KUKA KRL program: EPS_2_251825_SA15_A_20260116064058.src

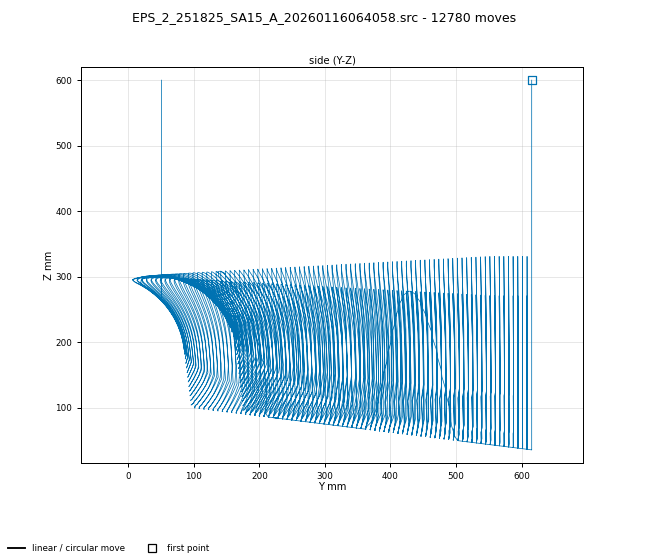
[picture p0: tool path of EPS_2_251825_SA15_A_20260116064058.src, 12780 of 12782 moves have a stored position in this frame; points joined in program order, loops and branches not executed]
&ACCESS RVP
&REL 4
&COMMENT QRS 19112012
&PARAM EDITMASK = *
DEF PART()
EXT BAS (BAS_COMMAND :IN,REAL :IN )
INT I
BAS (#INITMOV,0 )

;KUKA QRS Post kuka4.cps  Date:22-06-2017 !

File_ID=2977

QRS_PRE_INIT()

;Init var - Until changes are made in qrs_pre_init
Outlet_Square_prg=0
Inlet_1_Square_prg=0
Inlet_2_Square_prg=0
Inlet_3_Square_prg=0
Inlet_4_Square_prg=0
Inlet_5_Square_prg=0

Outlet_1={X 0.000, Y 551.740, Z 230.500, B 0.000, E1 0.000 }
Inlet_1={X 0.000, Y 556.010, Z 170.500, B 0.000, E1 166.000 }
Outlet_1_type=201
Inlet_1_type=201
;QRS#1=Sidecore dimensions
;QRS#2=200-8" PVC SDR 35
;QRS#3=200-8" PVC SDR 35
;QRS#4=
;QRS#5=
;QRS#6=
;QRS#7=
;QRS#8=
;QRS#9=12-08 PSX
;QRS#10=12-08 PSX
;QRS#11=
;QRS#12=
;QRS#13=
;QRS#14=
;QRS#15=
;QRS#16=1220x127x610 2'
;QRS#17=EPS Height
;QRS#18=331
;QRS#19=*
;QRS#20= UPDATED VERSION 22-06-2017
;QRS#21=*
Outlet_Square=0100
Inlet_1_Square=0100
Inlet_2_Square=0
Inlet_3_Square=0
Inlet_4_Square=0
Inlet_5_Square=0
Mill_Square=1
Outlet_Square_Prg=204
Inlet_1_Square_prg=204

QRS_INIT()

$ADVANCE=5

; T1
PTP {E1 173.614,E2 173.614}
PTP {X 0,Y 615.487,A -85,B 0,C 180,E1 173.614,E2 173.614,E3 0,E4 0,E5 0,E6 0}
QRS_SPEED_INIT()
LIN {X 0,Y 615.487,Z 600,A -85,B 0,C 180,E1 173.614,E2 173.614,E3 0,E4 0,E5 0,E6 0} C_VEL
LIN {X 0,Y 615.487,Z 45.866,A -85,B 0,C 180,E1 173.614,E2 173.614} C_VEL
LIN {X 0,Y 615.487,Z 37.686,A -85,B 0,C 180,E1 173.614,E2 173.614} C_VEL
LIN {X 0,Y 615.477,Z 35.686,A -85,B 0,C 180,E1 173.428,E2 173.428} C_VEL
LIN {X 0,Y 615.493,Z 35.696,A -85,B 0,C 180,E1 170.801,E2 170.801} C_VEL
LIN {X 0,Y 615.458,Z 35.693,A -85,B 0,C 180,E1 168.138,E2 168.138} C_VEL
LIN {X 0,Y 615.491,Z 35.686,A -85,B 0,C 180,E1 165.451,E2 165.451} C_VEL
LIN {X 0,Y 615.474,Z 35.697,A -85,B 0,C 180,E1 162.729,E2 162.729} C_VEL
LIN {X 0,Y 615.471,Z 35.688,A -85,B 0,C 180,E1 159.966,E2 159.966} C_VEL
LIN {X 0,Y 615.486,Z 35.701,A -85,B 0,C 180,E1 157.155,E2 157.155} C_VEL
LIN {X 0,Y 615.454,Z 35.691,A -85,B 0,C 180,E1 154.437,E2 154.437} C_VEL
LIN {X 0,Y 615.494,Z 35.698,A -85,B 0,C 180,E1 151.548,E2 151.548} C_VEL
LIN {X 0,Y 615.45,Z 35.694,A -85,B 0,C 180,E1 148.919,E2 148.919} C_VEL
LIN {X 0,Y 615.464,Z 35.69,A -85,B 0,C 180,E1 146.469,E2 146.469} C_VEL
LIN {X 0,Y 615.474,Z 35.698,A -85,B 0,C 180,E1 143.574,E2 143.574} C_VEL
LIN {X 0,Y 615.447,Z 35.693,A -85,B 0,C 180,E1 140.942,E2 140.942} C_VEL
LIN {X 0,Y 615.48,Z 35.69,A -85,B 0,C 180,E1 138.525,E2 138.525} C_VEL
LIN {X 0,Y 615.468,Z 35.698,A -85,B 0,C 180,E1 135.848,E2 135.848} C_VEL
LIN {X 0,Y 615.441,Z 35.694,A -85,B 0,C 180,E1 133.248,E2 133.248} C_VEL
LIN {X 0,Y 615.488,Z 35.694,A -85,B 0,C 180,E1 130.606,E2 130.606} C_VEL
LIN {X 0,Y 615.451,Z 35.698,A -85,B 0,C 180,E1 128.007,E2 128.007} C_VEL
LIN {X 0,Y 615.435,Z 35.695,A -85,B 0,C 180,E1 125.619,E2 125.619} C_VEL
LIN {X 0,Y 615.458,Z 35.694,A -85,B 0,C 180,E1 123.238,E2 123.238} C_VEL
LIN {X 0,Y 615.457,Z 35.707,A -85,B 0,C 180,E1 121.31,E2 121.31} C_VEL
LIN {X 0,Y 615.461,Z 51.527,A -85,B 0,C 180,E1 118.445,E2 118.445} C_VEL
LIN {X 0,Y 615.484,Z 60.763,A -85,B 0,C 180,E1 116.801,E2 116.801} C_VEL
LIN {X 0,Y 615.477,Z 167.66,A -85,B 0,C 180,E1 115.529,E2 115.529} C_VEL
LIN {X 0,Y 615.486,Z 180.477,A -85,B 0,C 180,E1 115.242,E2 115.242} C_VEL
LIN {X 0,Y 615.496,Z 193.451,A -85,B 0,C 180,E1 114.811,E2 114.811} C_VEL
LIN {X 0,Y 615.461,Z 205.297,A -85,B 0,C 180,E1 114.273,E2 114.273} C_VEL
LIN {X 0,Y 615.47,Z 215.754,A -85,B 0,C 180,E1 113.667,E2 113.667} C_VEL
LIN {X 0,Y 615.497,Z 225.992,A -85,B 0,C 180,E1 112.933,E2 112.933} C_VEL
LIN {X 0,Y 615.499,Z 235.079,A -85,B 0,C 180,E1 112.136,E2 112.136} C_VEL
LIN {X 0,Y 615.497,Z 243.269,A -85,B 0,C 180,E1 111.256,E2 111.256} C_VEL
LIN {X 0,Y 615.496,Z 250.555,A -85,B 0,C 180,E1 110.295,E2 110.295} C_VEL
LIN {X 0,Y 615.498,Z 256.431,A -85,B 0,C 180,E1 109.337,E2 109.337} C_VEL
LIN {X 0,Y 615.496,Z 261.553,A -85,B 0,C 180,E1 108.281,E2 108.281} C_VEL
LIN {X 0,Y 615.499,Z 265.263,A -85,B 0,C 180,E1 107.27,E2 107.27} C_VEL
LIN {X 0,Y 615.494,Z 267.552,A -85,B 0,C 180,E1 106.431,E2 106.431} C_VEL
LIN {X 0,Y 615.496,Z 269.625,A -85,B 0,C 180,E1 105.226,E2 105.226} C_VEL
LIN {X 0,Y 615.499,Z 270.387,A -85,B 0,C 180,E1 103.935,E2 103.935} C_VEL
LIN {X 0,Y 615.496,Z 270.103,A -85,B 0,C 180,E1 103.201,E2 103.201} C_VEL
LIN {X 0,Y 615.496,Z 269.443,A -85,B 0,C 180,E1 102.53,E2 102.53} C_VEL
LIN {X 0,Y 615.495,Z 268.377,A -85,B 0,C 180,E1 101.86,E2 101.86} C_VEL
LIN {X 0,Y 615.493,Z 266.032,A -85,B 0,C 180,E1 100.888,E2 100.888} C_VEL
LIN {X 0,Y 615.498,Z 262.525,A -85,B 0,C 180,E1 99.862,E2 99.862} C_VEL
LIN {X 0,Y 615.496,Z 258.019,A -85,B 0,C 180,E1 98.867,E2 98.867} C_VEL
LIN {X 0,Y 615.5,Z 251.196,A -85,B 0,C 180,E1 97.71,E2 97.71} C_VEL
LIN {X 0,Y 615.498,Z 243.968,A -85,B 0,C 180,E1 96.74,E2 96.74} C_VEL
LIN {X 0,Y 615.499,Z 236.316,A -85,B 0,C 180,E1 95.898,E2 95.898} C_VEL
LIN {X 0,Y 615.498,Z 227.254,A -85,B 0,C 180,E1 95.077,E2 95.077} C_VEL
LIN {X 0,Y 615.49,Z 217.212,A -85,B 0,C 180,E1 94.338,E2 94.338} C_VEL
LIN {X 0,Y 615.492,Z 206.13,A -85,B 0,C 180,E1 93.682,E2 93.682} C_VEL
LIN {X 0,Y 615.493,Z 195.661,A -85,B 0,C 180,E1 93.191,E2 93.191} C_VEL
LIN {X 0,Y 615.464,Z 183.105,A -85,B 0,C 180,E1 92.741,E2 92.741} C_VEL
LIN {X 0,Y 615.463,Z 170.568,A -85,B 0,C 180,E1 92.434,E2 92.434} C_VEL
LIN {X 0,Y 615.476,Z 152.905,A -85,B 0,C 180,E1 92.188,E2 92.188} C_VEL
LIN {X 0,Y 615.447,Z 60.667,A -85,B 0,C 180,E1 91.104,E2 91.104} C_VEL
LIN {X 0,Y 615.49,Z 45.411,A -85,B 0,C 180,E1 88.364,E2 88.364} C_VEL
LIN {X 0,Y 615.476,Z 35.689,A -85,B 0,C 180,E1 86.563,E2 86.563} C_VEL
LIN {X 0,Y 615.493,Z 35.682,A -85,B 0,C 180,E1 84.101,E2 84.101} C_VEL
LIN {X 0,Y 615.491,Z 35.698,A -85,B 0,C 180,E1 81.463,E2 81.463} C_VEL
LIN {X 0,Y 615.476,Z 35.688,A -85,B 0,C 180,E1 78.806,E2 78.806} C_VEL
LIN {X 0,Y 615.479,Z 35.689,A -85,B 0,C 180,E1 76.073,E2 76.073} C_VEL
LIN {X 0,Y 615.48,Z 35.697,A -85,B 0,C 180,E1 73.413,E2 73.413} C_VEL
LIN {X 0,Y 615.486,Z 35.684,A -85,B 0,C 180,E1 70.662,E2 70.662} C_VEL
LIN {X 0,Y 615.491,Z 35.701,A -85,B 0,C 180,E1 67.864,E2 67.864} C_VEL
LIN {X 0,Y 615.486,Z 35.684,A -85,B 0,C 180,E1 65.008,E2 65.008} C_VEL
LIN {X 0,Y 615.485,Z 35.701,A -85,B 0,C 180,E1 62.085,E2 62.085} C_VEL
LIN {X 0,Y 615.48,Z 35.695,A -85,B 0,C 180,E1 59.839,E2 59.839} C_VEL
LIN {X 0,Y 615.473,Z 35.689,A -85,B 0,C 180,E1 57.541,E2 57.541} C_VEL
LIN {X 0,Y 615.496,Z 35.681,A -85,B 0,C 180,E1 55.185,E2 55.185} C_VEL
LIN {X 0,Y 615.482,Z 35.692,A -85,B 0,C 180,E1 52.757,E2 52.757} C_VEL
LIN {X 0,Y 615.473,Z 35.691,A -85,B 0,C 180,E1 49.913,E2 49.913} C_VEL
LIN {X 0,Y 615.482,Z 35.685,A -85,B 0,C 180,E1 47.646,E2 47.646} C_VEL
LIN {X 0,Y 615.481,Z 35.694,A -85,B 0,C 180,E1 44.931,E2 44.931} C_VEL
LIN {X 0,Y 615.473,Z 35.689,A -85,B 0,C 180,E1 42.078,E2 42.078} C_VEL
LIN {X 0,Y 615.493,Z 35.682,A -85,B 0,C 180,E1 39.75,E2 39.75} C_VEL
LIN {X 0,Y 615.486,Z 35.702,A -85,B 0,C 180,E1 36.936,E2 36.936} C_VEL
LIN {X 0,Y 615.478,Z 35.695,A -85,B 0,C 180,E1 34.699,E2 34.699} C_VEL
LIN {X 0,Y 615.471,Z 35.688,A -85,B 0,C 180,E1 32.328,E2 32.328} C_VEL
LIN {X 0,Y 615.488,Z 35.686,A -85,B 0,C 180,E1 29.795,E2 29.795} C_VEL
LIN {X 0,Y 615.482,Z 35.697,A -85,B 0,C 180,E1 27.044,E2 27.044} C_VEL
LIN {X 0,Y 615.487,Z 35.683,A -85,B 0,C 180,E1 24.272,E2 24.272} C_VEL
LIN {X 0,Y 615.498,Z 35.7,A -85,B 0,C 180,E1 21.432,E2 21.432} C_VEL
LIN {X 0,Y 615.482,Z 35.685,A -85,B 0,C 180,E1 18.603,E2 18.603} C_VEL
LIN {X 0,Y 615.488,Z 35.694,A -85,B 0,C 180,E1 15.905,E2 15.905} C_VEL
LIN {X 0,Y 615.47,Z 35.691,A -85,B 0,C 180,E1 13.202,E2 13.202} C_VEL
LIN {X 0,Y 615.488,Z 35.685,A -85,B 0,C 180,E1 10.527,E2 10.527} C_VEL
LIN {X 0,Y 615.486,Z 35.701,A -85,B 0,C 180,E1 7.876,E2 7.876} C_VEL
LIN {X 0,Y 615.472,Z 35.688,A -85,B 0,C 180,E1 5.242,E2 5.242} C_VEL
LIN {X 0,Y 615.487,Z 35.688,A -85,B 0,C 180,E1 2.618,E2 2.618} C_VEL
LIN {X 0,Y 615.482,Z 35.697,A -85,B 0,C 180,E1 0,E2 0} C_VEL
LIN {X 0,Y 615.476,Z 35.686,A -85,B 0,C 180,E1 -2.618,E2 -2.618} C_VEL
LIN {X 0,Y 615.487,Z 35.691,A -85,B 0,C 180,E1 -5.241,E2 -5.241} C_VEL
LIN {X 0,Y 615.473,Z 35.695,A -85,B 0,C 180,E1 -7.876,E2 -7.876} C_VEL
LIN {X 0,Y 615.484,Z 35.684,A -85,B 0,C 180,E1 -10.527,E2 -10.527} C_VEL
LIN {X 0,Y 615.493,Z 35.697,A -85,B 0,C 180,E1 -13.201,E2 -13.201} C_VEL
LIN {X 0,Y 615.467,Z 35.69,A -85,B 0,C 180,E1 -15.906,E2 -15.906} C_VEL
LIN {X 0,Y 615.489,Z 35.688,A -85,B 0,C 180,E1 -18.646,E2 -18.646} C_VEL
LIN {X 0,Y 615.471,Z 35.694,A -85,B 0,C 180,E1 -21.432,E2 -21.432} C_VEL
LIN {X 0,Y 615.49,Z 35.685,A -85,B 0,C 180,E1 -24.272,E2 -24.272} C_VEL
LIN {X 0,Y 615.472,Z 35.695,A -85,B 0,C 180,E1 -27.178,E2 -27.178} C_VEL
LIN {X 0,Y 615.481,Z 35.685,A -85,B 0,C 180,E1 -29.793,E2 -29.793} C_VEL
LIN {X 0,Y 615.49,Z 35.696,A -85,B 0,C 180,E1 -32.457,E2 -32.457} C_VEL
LIN {X 0,Y 615.478,Z 35.697,A -85,B 0,C 180,E1 -34.816,E2 -34.816} C_VEL
LIN {X 0,Y 615.466,Z 35.689,A -85,B 0,C 180,E1 -37.244,E2 -37.244} C_VEL
LIN {X 0,Y 615.487,Z 35.693,A -85,B 0,C 180,E1 -40.089,E2 -40.089} C_VEL
LIN {X 0,Y 615.495,Z 35.699,A -85,B 0,C 180,E1 -42.353,E2 -42.353} C_VEL
LIN {X 0,Y 615.468,Z 35.688,A -85,B 0,C 180,E1 -45.071,E2 -45.071} C_VEL
LIN {X 0,Y 615.491,Z 35.695,A -85,B 0,C 180,E1 -47.92,E2 -47.92} C_VEL
LIN {X 0,Y 615.478,Z 35.697,A -85,B 0,C 180,E1 -50.249,E2 -50.249} C_VEL
LIN {X 0,Y 615.478,Z 35.686,A -85,B 0,C 180,E1 -53.065,E2 -53.065} C_VEL
LIN {X 0,Y 615.485,Z 35.698,A -85,B 0,C 180,E1 -55.978,E2 -55.978} C_VEL
LIN {X 0,Y 615.461,Z 35.693,A -85,B 0,C 180,E1 -58.313,E2 -58.313} C_VEL
LIN {X 0,Y 615.469,Z 35.688,A -85,B 0,C 180,E1 -60.593,E2 -60.593} C_VEL
LIN {X 0,Y 615.492,Z 35.702,A -85,B 0,C 180,E1 -63.556,E2 -63.556} C_VEL
LIN {X 0,Y 615.463,Z 35.693,A -85,B 0,C 180,E1 -65.997,E2 -65.997} C_VEL
LIN {X 0,Y 615.484,Z 35.871,A -85,B 0,C 180,E1 -66.711,E2 -66.711} C_VEL
LIN {X 0,Y 615.45,Z 57.104,A -85,B 0,C 180,E1 -69.453,E2 -69.453} C_VEL
LIN {X 0,Y 615.489,Z 77.473,A -85,B 0,C 180,E1 -72.043,E2 -72.043} C_VEL
LIN {X 0,Y 615.495,Z 99.259,A -85,B 0,C 180,E1 -74.774,E2 -74.774} C_VEL
LIN {X 0,Y 615.459,Z 118.133,A -85,B 0,C 180,E1 -77.113,E2 -77.113} C_VEL
LIN {X 0,Y 615.491,Z 226.817,A -85,B 0,C 180,E1 -78.411,E2 -78.411} C_VEL
LIN {X 0,Y 615.484,Z 239.337,A -85,B 0,C 180,E1 -78.682,E2 -78.682} C_VEL
LIN {X 0,Y 615.49,Z 252.593,A -85,B 0,C 180,E1 -79.112,E2 -79.112} C_VEL
LIN {X 0,Y 615.473,Z 264.475,A -85,B 0,C 180,E1 -79.639,E2 -79.639} C_VEL
LIN {X 0,Y 615.49,Z 275.991,A -85,B 0,C 180,E1 -80.304,E2 -80.304} C_VEL
LIN {X 0,Y 615.499,Z 286.338,A -85,B 0,C 180,E1 -81.05,E2 -81.05} C_VEL
LIN {X 0,Y 615.497,Z 294.809,A -85,B 0,C 180,E1 -81.794,E2 -81.794} C_VEL
LIN {X 0,Y 615.498,Z 302.604,A -85,B 0,C 180,E1 -82.619,E2 -82.619} C_VEL
LIN {X 0,Y 615.496,Z 310.201,A -85,B 0,C 180,E1 -83.608,E2 -83.608} C_VEL
LIN {X 0,Y 615.498,Z 317.203,A -85,B 0,C 180,E1 -84.759,E2 -84.759} C_VEL
LIN {X 0,Y 615.493,Z 321.85,A -85,B 0,C 180,E1 -85.743,E2 -85.743} C_VEL
LIN {X 0,Y 615.494,Z 325.398,A -85,B 0,C 180,E1 -86.727,E2 -86.727} C_VEL
LIN {X 0,Y 615.497,Z 327.232,A -85,B 0,C 180,E1 -87.382,E2 -87.382} C_VEL
LIN {X 0,Y 615.5,Z 328.607,A -85,B 0,C 180,E1 -88.037,E2 -88.037} C_VEL
LIN {X 0,Y 615.496,Z 330.173,A -85,B 0,C 180,E1 -89.346,E2 -89.346} C_VEL
LIN {X 0,Y 615.494,Z 330.389,A -85,B 0,C 180,E1 -90,E2 -90} C_VEL
LIN {X 0,Y 615.495,Z 329.58,A -85,B 0,C 180,E1 -91.308,E2 -91.308} C_VEL
LIN {X 0,Y 615.5,Z 328.608,A -85,B 0,C 180,E1 -91.963,E2 -91.963} C_VEL
LIN {X 0,Y 615.497,Z 327.234,A -85,B 0,C 180,E1 -92.618,E2 -92.618} C_VEL
LIN {X 0,Y 615.496,Z 324.35,A -85,B 0,C 180,E1 -93.6,E2 -93.6} C_VEL
LIN {X 0,Y 615.498,Z 320.442,A -85,B 0,C 180,E1 -94.584,E2 -94.584} C_VEL
LIN {X 0,Y 615.499,Z 315.406,A -85,B 0,C 180,E1 -95.569,E2 -95.569} C_VEL
LIN {X 0,Y 615.497,Z 308.869,A -85,B 0,C 180,E1 -96.583,E2 -96.583} C_VEL
LIN {X 0,Y 615.497,Z 301.135,A -85,B 0,C 180,E1 -97.545,E2 -97.545} C_VEL
LIN {X 0,Y 615.498,Z 293.048,A -85,B 0,C 180,E1 -98.371,E2 -98.371} C_VEL
LIN {X 0,Y 615.499,Z 283.171,A -85,B 0,C 180,E1 -99.198,E2 -99.198} C_VEL
LIN {X 0,Y 615.48,Z 271.987,A -85,B 0,C 180,E1 -99.945,E2 -99.945} C_VEL
LIN {X 0,Y 615.48,Z 261.029,A -85,B 0,C 180,E1 -100.527,E2 -100.527} C_VEL
LIN {X 0,Y 615.484,Z 248.48,A -85,B 0,C 180,E1 -101.04,E2 -101.04} C_VEL
LIN {X 0,Y 615.482,Z 236.078,A -85,B 0,C 180,E1 -101.401,E2 -101.401} C_VEL
LIN {X 0,Y 615.494,Z 222.483,A -85,B 0,C 180,E1 -101.652,E2 -101.652} C_VEL
LIN {X 0,Y 615.459,Z 118.137,A -85,B 0,C 180,E1 -102.887,E2 -102.887} C_VEL
LIN {X 0,Y 615.479,Z 95.179,A -85,B 0,C 180,E1 -105.735,E2 -105.735} C_VEL
LIN {X 0,Y 615.474,Z 73.671,A -85,B 0,C 180,E1 -108.438,E2 -108.438} C_VEL
LIN {X 0,Y 615.491,Z 51.569,A -85,B 0,C 180,E1 -111.256,E2 -111.256} C_VEL
LIN {X 0,Y 615.485,Z 35.685,A -85,B 0,C 180,E1 -113.333,E2 -113.333} C_VEL
LIN {X 0,Y 615.464,Z 35.69,A -85,B 0,C 180,E1 -115.716,E2 -115.716} C_VEL
LIN {X 0,Y 615.494,Z 35.697,A -85,B 0,C 180,E1 -118.451,E2 -118.451} C_VEL
LIN {X 0,Y 615.481,Z 35.685,A -85,B 0,C 180,E1 -121.085,E2 -121.085} C_VEL
LIN {X 0,Y 615.467,Z 35.691,A -85,B 0,C 180,E1 -123.531,E2 -123.531} C_VEL
LIN {X 0,Y 615.483,Z 35.697,A -85,B 0,C 180,E1 -125.833,E2 -125.833} C_VEL
LIN {X 0,Y 615.486,Z 35.698,A -85,B 0,C 180,E1 -128.068,E2 -128.068} C_VEL
LIN {X 0,Y 615.486,Z 35.685,A -85,B 0,C 180,E1 -130.606,E2 -130.606} C_VEL
LIN {X 0,Y 615.473,Z 35.692,A -85,B 0,C 180,E1 -133.245,E2 -133.245} C_VEL
LIN {X 0,Y 615.484,Z 35.691,A -85,B 0,C 180,E1 -136.002,E2 -136.002} C_VEL
LIN {X 0,Y 615.486,Z 35.684,A -85,B 0,C 180,E1 -138.526,E2 -138.526} C_VEL
LIN {X 0,Y 615.48,Z 35.695,A -85,B 0,C 180,E1 -141.095,E2 -141.095} C_VEL
LIN {X 0,Y 615.483,Z 35.694,A -85,B 0,C 180,E1 -143.575,E2 -143.575} C_VEL
LIN {X 0,Y 615.485,Z 35.685,A -85,B 0,C 180,E1 -145.978,E2 -145.978} C_VEL
LIN {X 0,Y 615.482,Z 35.699,A -85,B 0,C 180,E1 -148.914,E2 -148.914} C_VEL
LIN {X 0,Y 615.479,Z 35.688,A -85,B 0,C 180,E1 -151.55,E2 -151.55} C_VEL
LIN {X 0,Y 615.48,Z 35.689,A -85,B 0,C 180,E1 -154.284,E2 -154.284} C_VEL
LIN {X 0,Y 615.484,Z 35.694,A -85,B 0,C 180,E1 -156.444,E2 -156.444} C_VEL
LIN {X 0,Y 615.476,Z 35.688,A -85,B 0,C 180,E1 -159.269,E2 -159.269} C_VEL
LIN {X 0,Y 615.483,Z 35.69,A -85,B 0,C 180,E1 -162.043,E2 -162.043} C_VEL
LIN {X 0,Y 615.475,Z 35.693,A -85,B 0,C 180,E1 -164.774,E2 -164.774} C_VEL
LIN {X 0,Y 615.489,Z 35.684,A -85,B 0,C 180,E1 -167.47,E2 -167.47} C_VEL
LIN {X 0,Y 615.499,Z 35.7,A -85,B 0,C 180,E1 -170.138,E2 -170.138} C_VEL
LIN {X 0,Y 615.471,Z 35.689,A -85,B 0,C 180,E1 -172.784,E2 -172.784} C_VEL
LIN {X 0,Y 615.488,Z 35.688,A -85,B 0,C 180,E1 -175.416,E2 -175.416} C_VEL
LIN {X 0,Y 615.481,Z 35.697,A -85,B 0,C 180,E1 -178.037,E2 -178.037} C_VEL
LIN {X 0,Y 615.474,Z 35.687,A -85,B 0,C 180,E1 -180.654,E2 -180.654} C_VEL
LIN {X 0,Y 615.487,Z 35.692,A -85,B 0,C 180,E1 -183.273,E2 -183.273} C_VEL
LIN {X 0,Y 615.467,Z 35.695,A -85,B 0,C 180,E1 -185.899,E2 -185.899} C_VEL
LIN {X 0,Y 615.477,Z 35.686,A -85,B 0,C 180,E1 -186.572,E2 -186.572} C_VEL
LIN {X 0,Y 614.812,Z 35.842,A -85,B 0,C 180,E1 -187.118,E2 -187.118} C_VEL
LIN {X 0,Y 611.99,Z 36.249,A -85,B 0,C 180,E1 -188.004,E2 -188.004} C_VEL
LIN {X 0,Y 609.597,Z 36.565,A -85,B 0,C 180,E1 -188.717,E2 -188.717} C_VEL
LIN {X 0,Y 608.552,Z 36.686,A -85,B 0,C 180,E1 -189.266,E2 -189.266} C_VEL
LIN {X 0,Y 608.457,Z 36.694,A -85,B 0,C 180,E1 -189.452,E2 -189.452} C_VEL
LIN {X 0,Y 608.443,Z 36.69,A -85,B 0,C 180,E1 -192,E2 -192} C_VEL
LIN {X 0,Y 608.478,Z 36.689,A -85,B 0,C 180,E1 -194.721,E2 -194.721} C_VEL
LIN {X 0,Y 608.438,Z 36.692,A -85,B 0,C 180,E1 -197.477,E2 -197.477} C_VEL
LIN {X 0,Y 608.434,Z 36.691,A -85,B 0,C 180,E1 -199.571,E2 -199.571} C_VEL
LIN {X 0,Y 608.45,Z 36.688,A -85,B 0,C 180,E1 -201.693,E2 -201.693} C_VEL
LIN {X 0,Y 608.449,Z 36.696,A -85,B 0,C 180,E1 -204.572,E2 -204.572} C_VEL
LIN {X 0,Y 608.433,Z 36.69,A -85,B 0,C 180,E1 -207.519,E2 -207.519} C_VEL
LIN {X 0,Y 608.464,Z 36.689,A -85,B 0,C 180,E1 -209.972,E2 -209.972} C_VEL
LIN {X 0,Y 608.441,Z 36.692,A -85,B 0,C 180,E1 -212.881,E2 -212.881} C_VEL
LIN {X 0,Y 608.424,Z 36.691,A -85,B 0,C 180,E1 -215.279,E2 -215.279} C_VEL
LIN {X 0,Y 608.469,Z 36.694,A -85,B 0,C 180,E1 -218.241,E2 -218.241} C_VEL
LIN {X 0,Y 608.444,Z 36.69,A -85,B 0,C 180,E1 -221.341,E2 -221.341} C_VEL
LIN {X 0,Y 608.437,Z 36.694,A -85,B 0,C 180,E1 -224.262,E2 -224.262} C_VEL
LIN {X 0,Y 608.435,Z 36.69,A -85,B 0,C 180,E1 -226.695,E2 -226.695} C_VEL
LIN {X 0,Y 608.417,Z 36.693,A -85,B 0,C 180,E1 -228.821,E2 -228.821} C_VEL
LIN {X 0,Y 608.444,Z 36.696,A -85,B 0,C 180,E1 -231.763,E2 -231.763} C_VEL
LIN {X 0,Y 608.433,Z 36.693,A -85,B 0,C 180,E1 -233.957,E2 -233.957} C_VEL
LIN {X 0,Y 608.412,Z 36.693,A -85,B 0,C 180,E1 -236.326,E2 -236.326} C_VEL
LIN {X 0,Y 608.47,Z 36.892,A -85,B 0,C 180,E1 -238.684,E2 -238.684} C_VEL
LIN {X 0,Y 608.455,Z 51.687,A -85,B 0,C 180,E1 -241.384,E2 -241.384} C_VEL
LIN {X 0,Y 608.479,Z 61.04,A -85,B 0,C 180,E1 -243.051,E2 -243.051} C_VEL
LIN {X 0,Y 608.535,Z 167.622,A -85,B 0,C 180,E1 -244.334,E2 -244.334} C_VEL
LIN {X 0,Y 608.531,Z 181.356,A -85,B 0,C 180,E1 -244.649,E2 -244.649} C_VEL
LIN {X 0,Y 608.524,Z 193.704,A -85,B 0,C 180,E1 -245.068,E2 -245.068} C_VEL
LIN {X 0,Y 608.488,Z 205.702,A -85,B 0,C 180,E1 -245.621,E2 -245.621} C_VEL
LIN {X 0,Y 608.477,Z 217.729,A -85,B 0,C 180,E1 -246.337,E2 -246.337} C_VEL
LIN {X 0,Y 608.493,Z 228.507,A -85,B 0,C 180,E1 -247.148,E2 -247.148} C_VEL
LIN {X 0,Y 608.456,Z 237.187,A -85,B 0,C 180,E1 -247.952,E2 -247.952} C_VEL
LIN {X 0,Y 608.449,Z 245.112,A -85,B 0,C 180,E1 -248.841,E2 -248.841} C_VEL
LIN {X 0,Y 608.438,Z 252.786,A -85,B 0,C 180,E1 -249.902,E2 -249.902} C_VEL
LIN {X 0,Y 608.44,Z 257.883,A -85,B 0,C 180,E1 -250.78,E2 -250.78} C_VEL
LIN {X 0,Y 608.43,Z 262.75,A -85,B 0,C 180,E1 -251.828,E2 -251.828} C_VEL
LIN {X 0,Y 608.453,Z 266.389,A -85,B 0,C 180,E1 -252.87,E2 -252.87} C_VEL
LIN {X 0,Y 608.433,Z 268.924,A -85,B 0,C 180,E1 -253.906,E2 -253.906} C_VEL
LIN {X 0,Y 608.42,Z 270.033,A -85,B 0,C 180,E1 -254.593,E2 -254.593} C_VEL
LIN {X 0,Y 608.418,Z 270.71,A -85,B 0,C 180,E1 -255.278,E2 -255.278} C_VEL
LIN {X 0,Y 608.446,Z 270.994,A -85,B 0,C 180,E1 -255.994,E2 -255.994} C_VEL
LIN {X 0,Y 608.439,Z 270.828,A -85,B 0,C 180,E1 -256.643,E2 -256.643} C_VEL
LIN {X 0,Y 608.44,Z 269.252,A -85,B 0,C 180,E1 -258,E2 -258} C_VEL
LIN {X 0,Y 608.422,Z 266.804,A -85,B 0,C 180,E1 -259.07,E2 -259.07} C_VEL
LIN {X 0,Y 608.437,Z 263.663,A -85,B 0,C 180,E1 -260.023,E2 -260.023} C_VEL
LIN {X 0,Y 608.447,Z 259.295,A -85,B 0,C 180,E1 -261.029,E2 -261.029} C_VEL
LIN {X 0,Y 608.439,Z 253.74,A -85,B 0,C 180,E1 -262.033,E2 -262.033} C_VEL
LIN {X 0,Y 608.466,Z 246.824,A -85,B 0,C 180,E1 -263.034,E2 -263.034} C_VEL
LIN {X 0,Y 608.455,Z 238.208,A -85,B 0,C 180,E1 -264.033,E2 -264.033} C_VEL
LIN {X 0,Y 608.483,Z 229.406,A -85,B 0,C 180,E1 -264.865,E2 -264.865} C_VEL
LIN {X 0,Y 608.491,Z 218.616,A -85,B 0,C 180,E1 -265.695,E2 -265.695} C_VEL
LIN {X 0,Y 608.509,Z 207.761,A -85,B 0,C 180,E1 -266.358,E2 -266.358} C_VEL
LIN {X 0,Y 608.533,Z 195.693,A -85,B 0,C 180,E1 -266.938,E2 -266.938} C_VEL
LIN {X 0,Y 608.497,Z 183.08,A -85,B 0,C 180,E1 -267.394,E2 -267.394} C_VEL
LIN {X 0,Y 608.527,Z 170.432,A -85,B 0,C 180,E1 -267.704,E2 -267.704} C_VEL
LIN {X 0,Y 608.54,Z 152.663,A -85,B 0,C 180,E1 -267.953,E2 -267.953} C_VEL
LIN {X 0,Y 608.426,Z 60.861,A -85,B 0,C 180,E1 -269.049,E2 -269.049} C_VEL
LIN {X 0,Y 608.484,Z 46.461,A -85,B 0,C 180,E1 -271.655,E2 -271.655} C_VEL
LIN {X 0,Y 608.454,Z 36.689,A -85,B 0,C 180,E1 -273.477,E2 -273.477} C_VEL
LIN {X 0,Y 608.466,Z 36.687,A -85,B 0,C 180,E1 -275.967,E2 -275.967} C_VEL
LIN {X 0,Y 608.459,Z 36.698,A -85,B 0,C 180,E1 -278.636,E2 -278.636} C_VEL
LIN {X 0,Y 608.443,Z 36.689,A -85,B 0,C 180,E1 -281.325,E2 -281.325} C_VEL
LIN {X 0,Y 608.475,Z 36.689,A -85,B 0,C 180,E1 -284.038,E2 -284.038} C_VEL
LIN {X 0,Y 608.445,Z 36.692,A -85,B 0,C 180,E1 -286.784,E2 -286.784} C_VEL
LIN {X 0,Y 608.453,Z 36.689,A -85,B 0,C 180,E1 -289.571,E2 -289.571} C_VEL
LIN {X 0,Y 608.465,Z 36.691,A -85,B 0,C 180,E1 -292.476,E2 -292.476} C_VEL
LIN {X 0,Y 608.455,Z 36.69,A -85,B 0,C 180,E1 -294.571,E2 -294.571} C_VEL
LIN {X 0,Y 608.485,Z 36.684,A -85,B 0,C 180,E1 -297.207,E2 -297.207} C_VEL
LIN {X 0,Y 608.47,Z 36.695,A -85,B 0,C 180,E1 -299.971,E2 -299.971} C_VEL
LIN {X 0,Y 608.453,Z 36.688,A -85,B 0,C 180,E1 -302.88,E2 -302.88} C_VEL
LIN {X 0,Y 608.452,Z 36.691,A -85,B 0,C 180,E1 -305.277,E2 -305.277} C_VEL
LIN {X 0,Y 608.462,Z 36.695,A -85,B 0,C 180,E1 -307.747,E2 -307.747} C_VEL
LIN {X 0,Y 608.444,Z 36.689,A -85,B 0,C 180,E1 -310.327,E2 -310.327} C_VEL
LIN {X 0,Y 608.476,Z 36.693,A -85,B 0,C 180,E1 -313.309,E2 -313.309} C_VEL
LIN {X 0,Y 608.461,Z 36.687,A -85,B 0,C 180,E1 -316.129,E2 -316.129} C_VEL
LIN {X 0,Y 608.455,Z 36.691,A -85,B 0,C 180,E1 -318.823,E2 -318.823} C_VEL
LIN {X 0,Y 608.442,Z 36.695,A -85,B 0,C 180,E1 -321.409,E2 -321.409} C_VEL
LIN {X 0,Y 608.449,Z 36.688,A -85,B 0,C 180,E1 -323.954,E2 -323.954} C_VEL
LIN {X 0,Y 608.452,Z 36.689,A -85,B 0,C 180,E1 -326.328,E2 -326.328} C_VEL
LIN {X 0,Y 608.451,Z 36.696,A -85,B 0,C 180,E1 -328.732,E2 -328.732} C_VEL
LIN {X 0,Y 608.462,Z 36.688,A -85,B 0,C 180,E1 -331.382,E2 -331.382} C_VEL
LIN {X 0,Y 608.441,Z 36.69,A -85,B 0,C 180,E1 -333.964,E2 -333.964} C_VEL
LIN {X 0,Y 608.47,Z 36.688,A -85,B 0,C 180,E1 -336.155,E2 -336.155} C_VEL
LIN {X 0,Y 608.476,Z 36.691,A -85,B 0,C 180,E1 -338.308,E2 -338.308} C_VEL
LIN {X 0,Y 608.469,Z 36.686,A -85,B 0,C 180,E1 -341.285,E2 -341.285} C_VEL
LIN {X 0,Y 608.463,Z 36.69,A -85,B 0,C 180,E1 -343.906,E2 -343.906} C_VEL
LIN {X 0,Y 608.453,Z 36.692,A -85,B 0,C 180,E1 -346.643,E2 -346.643} C_VEL
LIN {X 0,Y 608.464,Z 36.687,A -85,B 0,C 180,E1 -349.35,E2 -349.35} C_VEL
LIN {X 0,Y 608.479,Z 36.694,A -85,B 0,C 180,E1 -352.033,E2 -352.033} C_VEL
LIN {X 0,Y 608.454,Z 36.688,A -85,B 0,C 180,E1 -354.698,E2 -354.698} C_VEL
LIN {X 0,Y 608.478,Z 36.687,A -85,B 0,C 180,E1 -357.352,E2 -357.352} C_VEL
LIN {X 0,Y 608.473,Z 36.692,A -85,B 0,C 180,E1 -360,E2 -360} C_VEL
LIN {X 0,Y 608.469,Z 36.686,A -85,B 0,C 180,E1 -362.648,E2 -362.648} C_VEL
LIN {X 0,Y 608.465,Z 36.691,A -85,B 0,C 180,E1 -365.302,E2 -365.302} C_VEL
LIN {X 0,Y 608.468,Z 36.689,A -85,B 0,C 180,E1 -367.967,E2 -367.967} C_VEL
LIN {X 0,Y 608.464,Z 36.687,A -85,B 0,C 180,E1 -370.65,E2 -370.65} C_VEL
LIN {X 0,Y 608.464,Z 36.696,A -85,B 0,C 180,E1 -373.356,E2 -373.356} C_VEL
LIN {X 0,Y 608.45,Z 36.688,A -85,B 0,C 180,E1 -376.094,E2 -376.094} C_VEL
LIN {X 0,Y 608.457,Z 36.693,A -85,B 0,C 180,E1 -378.87,E2 -378.87} C_VEL
LIN {X 0,Y 608.46,Z 36.688,A -85,B 0,C 180,E1 -381.692,E2 -381.692} C_VEL
LIN {X 0,Y 608.456,Z 36.692,A -85,B 0,C 180,E1 -384.571,E2 -384.571} C_VEL
LIN {X 0,Y 608.443,Z 36.69,A -85,B 0,C 180,E1 -387.518,E2 -387.518} C_VEL
LIN {X 0,Y 608.466,Z 36.687,A -85,B 0,C 180,E1 -389.971,E2 -389.971} C_VEL
LIN {X 0,Y 608.449,Z 36.694,A -85,B 0,C 180,E1 -392.88,E2 -392.88} C_VEL
LIN {X 0,Y 608.436,Z 36.691,A -85,B 0,C 180,E1 -395.278,E2 -395.278} C_VEL
LIN {X 0,Y 608.467,Z 36.693,A -85,B 0,C 180,E1 -398.24,E2 -398.24} C_VEL
LIN {X 0,Y 608.453,Z 36.688,A -85,B 0,C 180,E1 -401.341,E2 -401.341} C_VEL
LIN {X 0,Y 608.461,Z 36.697,A -85,B 0,C 180,E1 -404.264,E2 -404.264} C_VEL
LIN {X 0,Y 608.436,Z 36.69,A -85,B 0,C 180,E1 -407.039,E2 -407.039} C_VEL
LIN {X 0,Y 608.456,Z 36.692,A -85,B 0,C 180,E1 -409.697,E2 -409.697} C_VEL
LIN {X 0,Y 608.462,Z 36.692,A -85,B 0,C 180,E1 -412.253,E2 -412.253} C_VEL
LIN {X 0,Y 608.458,Z 36.688,A -85,B 0,C 180,E1 -415.094,E2 -415.094} C_VEL
LIN {X 0,Y 608.465,Z 36.694,A -85,B 0,C 180,E1 -417.905,E2 -417.905} C_VEL
LIN {X 0,Y 608.45,Z 36.69,A -85,B 0,C 180,E1 -420.219,E2 -420.219} C_VEL
LIN {X 0,Y 608.482,Z 36.685,A -85,B 0,C 180,E1 -422.793,E2 -422.793} C_VEL
LIN {X 0,Y 608.464,Z 36.692,A -85,B 0,C 180,E1 -425.851,E2 -425.851} C_VEL
LIN {X 0,Y 608.51,Z 36.895,A -85,B 0,C 180,E1 -426.563,E2 -426.563} C_VEL
LIN {X 0,Y 608.569,Z 54.295,A -85,B 0,C 180,E1 -428.845,E2 -428.845} C_VEL
LIN {X 0,Y 608.537,Z 74.958,A -85,B 0,C 180,E1 -431.507,E2 -431.507} C_VEL
LIN {X 0,Y 608.489,Z 96.602,A -85,B 0,C 180,E1 -434.251,E2 -434.251} C_VEL
LIN {X 0,Y 608.456,Z 118.353,A -85,B 0,C 180,E1 -436.972,E2 -436.972} C_VEL
LIN {X 0,Y 608.547,Z 226.935,A -85,B 0,C 180,E1 -438.276,E2 -438.276} C_VEL
LIN {X 0,Y 608.519,Z 240.209,A -85,B 0,C 180,E1 -438.571,E2 -438.571} C_VEL
LIN {X 0,Y 608.516,Z 252.614,A -85,B 0,C 180,E1 -438.982,E2 -438.982} C_VEL
LIN {X 0,Y 608.497,Z 264.63,A -85,B 0,C 180,E1 -439.519,E2 -439.519} C_VEL
LIN {X 0,Y 608.477,Z 276.194,A -85,B 0,C 180,E1 -440.191,E2 -440.191} C_VEL
LIN {X 0,Y 608.485,Z 286.591,A -85,B 0,C 180,E1 -440.946,E2 -440.946} C_VEL
LIN {X 0,Y 608.475,Z 295.109,A -85,B 0,C 180,E1 -441.699,E2 -441.699} C_VEL
LIN {X 0,Y 608.471,Z 302.958,A -85,B 0,C 180,E1 -442.534,E2 -442.534} C_VEL
LIN {X 0,Y 608.461,Z 310.286,A -85,B 0,C 180,E1 -443.484,E2 -443.484} C_VEL
LIN {X 0,Y 608.451,Z 315.865,A -85,B 0,C 180,E1 -444.365,E2 -444.365} C_VEL
LIN {X 0,Y 608.432,Z 320.949,A -85,B 0,C 180,E1 -445.362,E2 -445.362} C_VEL
LIN {X 0,Y 608.449,Z 324.895,A -85,B 0,C 180,E1 -446.357,E2 -446.357} C_VEL
LIN {X 0,Y 608.425,Z 327.808,A -85,B 0,C 180,E1 -447.352,E2 -447.352} C_VEL
LIN {X 0,Y 608.444,Z 329.201,A -85,B 0,C 180,E1 -448.014,E2 -448.014} C_VEL
LIN {X 0,Y 608.439,Z 330.783,A -85,B 0,C 180,E1 -449.338,E2 -449.338} C_VEL
LIN {X 0,Y 608.434,Z 331,A -85,B 0,C 180,E1 -450,E2 -450} C_VEL
LIN {X 0,Y 608.448,Z 330.184,A -85,B 0,C 180,E1 -451.323,E2 -451.323} C_VEL
LIN {X 0,Y 608.444,Z 329.202,A -85,B 0,C 180,E1 -451.986,E2 -451.986} C_VEL
LIN {X 0,Y 608.425,Z 327.81,A -85,B 0,C 180,E1 -452.648,E2 -452.648} C_VEL
LIN {X 0,Y 608.449,Z 324.897,A -85,B 0,C 180,E1 -453.642,E2 -453.642} C_VEL
LIN {X 0,Y 608.432,Z 320.951,A -85,B 0,C 180,E1 -454.638,E2 -454.638} C_VEL
LIN {X 0,Y 608.438,Z 314.878,A -85,B 0,C 180,E1 -455.801,E2 -455.801} C_VEL
LIN {X 0,Y 608.462,Z 308.237,A -85,B 0,C 180,E1 -456.799,E2 -456.799} C_VEL
LIN {X 0,Y 608.456,Z 299.991,A -85,B 0,C 180,E1 -457.8,E2 -457.8} C_VEL
LIN {X 0,Y 608.472,Z 291.539,A -85,B 0,C 180,E1 -458.636,E2 -458.636} C_VEL
LIN {X 0,Y 608.48,Z 281.095,A -85,B 0,C 180,E1 -459.473,E2 -459.473} C_VEL
LIN {X 0,Y 608.484,Z 270.761,A -85,B 0,C 180,E1 -460.145,E2 -460.145} C_VEL
LIN {X 0,Y 608.519,Z 259.266,A -85,B 0,C 180,E1 -460.74,E2 -460.74} C_VEL
LIN {X 0,Y 608.53,Z 246.894,A -85,B 0,C 180,E1 -461.225,E2 -461.225} C_VEL
LIN {X 0,Y 608.545,Z 233.45,A -85,B 0,C 180,E1 -461.596,E2 -461.596} C_VEL
LIN {X 0,Y 608.552,Z 221.105,A -85,B 0,C 180,E1 -461.808,E2 -461.808} C_VEL
LIN {X 0,Y 608.445,Z 118.272,A -85,B 0,C 180,E1 -463.038,E2 -463.038} C_VEL
LIN {X 0,Y 608.495,Z 95.242,A -85,B 0,C 180,E1 -465.92,E2 -465.92} C_VEL
LIN {X 0,Y 608.537,Z 74.96,A -85,B 0,C 180,E1 -468.493,E2 -468.493} C_VEL
LIN {X 0,Y 608.569,Z 54.299,A -85,B 0,C 180,E1 -471.154,E2 -471.154} C_VEL
LIN {X 0,Y 608.511,Z 36.899,A -85,B 0,C 180,E1 -473.436,E2 -473.436} C_VEL
LIN {X 0,Y 608.449,Z 36.691,A -85,B 0,C 180,E1 -473.845,E2 -473.845} C_VEL
LIN {X 0,Y 608.459,Z 36.691,A -85,B 0,C 180,E1 -476.773,E2 -476.773} C_VEL
LIN {X 0,Y 608.466,Z 36.687,A -85,B 0,C 180,E1 -479.02,E2 -479.02} C_VEL
LIN {X 0,Y 608.443,Z 36.689,A -85,B 0,C 180,E1 -481.317,E2 -481.317} C_VEL
LIN {X 0,Y 608.445,Z 36.693,A -85,B 0,C 180,E1 -483.731,E2 -483.731} C_VEL
LIN {X 0,Y 608.477,Z 36.694,A -85,B 0,C 180,E1 -486.09,E2 -486.09} C_VEL
LIN {X 0,Y 608.467,Z 36.687,A -85,B 0,C 180,E1 -488.588,E2 -488.588} C_VEL
LIN {X 0,Y 608.452,Z 36.691,A -85,B 0,C 180,E1 -491.341,E2 -491.341} C_VEL
LIN {X 0,Y 608.45,Z 36.69,A -85,B 0,C 180,E1 -494.263,E2 -494.263} C_VEL
LIN {X 0,Y 608.442,Z 36.692,A -85,B 0,C 180,E1 -497.039,E2 -497.039} C_VEL
LIN {X 0,Y 608.451,Z 36.694,A -85,B 0,C 180,E1 -499.696,E2 -499.696} C_VEL
LIN {X 0,Y 608.465,Z 36.686,A -85,B 0,C 180,E1 -502.253,E2 -502.253} C_VEL
LIN {X 0,Y 608.487,Z 36.692,A -85,B 0,C 180,E1 -505.089,E2 -505.089} C_VEL
LIN {X 0,Y 608.461,Z 36.687,A -85,B 0,C 180,E1 -507.905,E2 -507.905} C_VEL
LIN {X 0,Y 608.47,Z 36.686,A -85,B 0,C 180,E1 -510.221,E2 -510.221} C_VEL
LIN {X 0,Y 608.481,Z 36.693,A -85,B 0,C 180,E1 -512.791,E2 -512.791} C_VEL
LIN {X 0,Y 608.453,Z 36.689,A -85,B 0,C 180,E1 -515.429,E2 -515.429} C_VEL
LIN {X 0,Y 608.473,Z 36.69,A -85,B 0,C 180,E1 -518.309,E2 -518.309} C_VEL
LIN {X 0,Y 608.468,Z 36.687,A -85,B 0,C 180,E1 -521.284,E2 -521.284} C_VEL
LIN {X 0,Y 608.461,Z 36.689,A -85,B 0,C 180,E1 -523.906,E2 -523.906} C_VEL
LIN {X 0,Y 608.454,Z 36.692,A -85,B 0,C 180,E1 -526.643,E2 -526.643} C_VEL
LIN {X 0,Y 608.464,Z 36.687,A -85,B 0,C 180,E1 -529.35,E2 -529.35} C_VEL
LIN {X 0,Y 608.478,Z 36.694,A -85,B 0,C 180,E1 -532.033,E2 -532.033} C_VEL
LIN {X 0,Y 608.453,Z 36.689,A -85,B 0,C 180,E1 -534.698,E2 -534.698} C_VEL
LIN {X 0,Y 608.478,Z 36.687,A -85,B 0,C 180,E1 -537.352,E2 -537.352} C_VEL
LIN {X 0,Y 608.469,Z 36.692,A -85,B 0,C 180,E1 -540,E2 -540} C_VEL
LIN {X 0,Y 608.467,Z 36.686,A -85,B 0,C 180,E1 -542.648,E2 -542.648} C_VEL
LIN {X 0,Y 608.467,Z 36.693,A -85,B 0,C 180,E1 -545.302,E2 -545.302} C_VEL
LIN {X 0,Y 608.432,Z 36.692,A -85,B 0,C 180,E1 -547.968,E2 -547.968} C_VEL
LIN {X 0,Y 608.457,Z 36.694,A -85,B 0,C 180,E1 -549.452,E2 -549.452} C_VEL
LIN {X 0,Y 607.764,Z 36.776,A -85,B 0,C 180,E1 -550.005,E2 -550.005} C_VEL
LIN {X 0,Y 604.901,Z 37.134,A -85,B 0,C 180,E1 -550.902,E2 -550.902} C_VEL
LIN {X 0,Y 602.503,Z 37.433,A -85,B 0,C 180,E1 -551.624,E2 -551.624} C_VEL
LIN {X 0,Y 601.482,Z 37.556,A -85,B 0,C 180,E1 -552.18,E2 -552.18} C_VEL
LIN {X 0,Y 601.402,Z 37.566,A -85,B 0,C 180,E1 -552.369,E2 -552.369} C_VEL
LIN {X 0,Y 601.429,Z 37.569,A -85,B 0,C 180,E1 -554.897,E2 -554.897} C_VEL
LIN {X 0,Y 601.428,Z 37.573,A -85,B 0,C 180,E1 -556.986,E2 -556.986} C_VEL
LIN {X 0,Y 601.394,Z 37.567,A -85,B 0,C 180,E1 -559.81,E2 -559.81} C_VEL
LIN {X 0,Y 601.404,Z 37.566,A -85,B 0,C 180,E1 -561.96,E2 -561.96} C_VEL
LIN {X 0,Y 601.433,Z 37.566,A -85,B 0,C 180,E1 -564.293,E2 -564.293} C_VEL
LIN {X 0,Y 601.395,Z 37.57,A -85,B 0,C 180,E1 -567.114,E2 -567.114} C_VEL
LIN {X 0,Y 601.395,Z 37.567,A -85,B 0,C 180,E1 -569.395,E2 -569.395} C_VEL
LIN {X 0,Y 601.398,Z 37.568,A -85,B 0,C 180,E1 -571.728,E2 -571.728} C_VEL
LIN {X 0,Y 601.414,Z 37.572,A -85,B 0,C 180,E1 -574.12,E2 -574.12} C_VEL
LIN {X 0,Y 601.387,Z 37.572,A -85,B 0,C 180,E1 -576.585,E2 -576.585} C_VEL
LIN {X 0,Y 601.39,Z 37.568,A -85,B 0,C 180,E1 -579.129,E2 -579.129} C_VEL
LIN {X 0,Y 601.418,Z 37.57,A -85,B 0,C 180,E1 -581.766,E2 -581.766} C_VEL
LIN {X 0,Y 601.398,Z 37.568,A -85,B 0,C 180,E1 -584.533,E2 -584.533} C_VEL
LIN {X 0,Y 601.411,Z 37.57,A -85,B 0,C 180,E1 -587.41,E2 -587.41} C_VEL
LIN {X 0,Y 601.395,Z 37.571,A -85,B 0,C 180,E1 -590.004,E2 -590.004} C_VEL
LIN {X 0,Y 601.396,Z 37.567,A -85,B 0,C 180,E1 -592.624,E2 -592.624} C_VEL
LIN {X 0,Y 601.413,Z 37.57,A -85,B 0,C 180,E1 -595.068,E2 -595.068} C_VEL
LIN {X 0,Y 601.418,Z 37.573,A -85,B 0,C 180,E1 -597.484,E2 -597.484} C_VEL
LIN {X 0,Y 601.396,Z 37.638,A -85,B 0,C 180,E1 -598.612,E2 -598.612} C_VEL
LIN {X 0,Y 601.415,Z 52.581,A -85,B 0,C 180,E1 -601.373,E2 -601.373} C_VEL
LIN {X 0,Y 601.411,Z 60.864,A -85,B 0,C 180,E1 -602.887,E2 -602.887} C_VEL
LIN {X 0,Y 601.66,Z 70.655,A -85,B 0,C 180,E1 -603.017,E2 -603.017} C_VEL
LIN {X 0,Y 601.598,Z 167.413,A -85,B 0,C 180,E1 -604.193,E2 -604.193} C_VEL
LIN {X 0,Y 601.577,Z 181.014,A -85,B 0,C 180,E1 -604.505,E2 -604.505} C_VEL
LIN {X 0,Y 601.542,Z 193.812,A -85,B 0,C 180,E1 -604.943,E2 -604.943} C_VEL
LIN {X 0,Y 601.477,Z 206.455,A -85,B 0,C 180,E1 -605.539,E2 -605.539} C_VEL
LIN {X 0,Y 601.457,Z 217.793,A -85,B 0,C 180,E1 -606.226,E2 -606.226} C_VEL
LIN {X 0,Y 601.451,Z 228.548,A -85,B 0,C 180,E1 -607.046,E2 -607.046} C_VEL
LIN {X 0,Y 601.416,Z 237.246,A -85,B 0,C 180,E1 -607.863,E2 -607.863} C_VEL
LIN {X 0,Y 601.384,Z 246.21,A -85,B 0,C 180,E1 -608.893,E2 -608.893} C_VEL
LIN {X 0,Y 601.37,Z 253.892,A -85,B 0,C 180,E1 -610.012,E2 -610.012} C_VEL
LIN {X 0,Y 601.347,Z 260.258,A -85,B 0,C 180,E1 -611.202,E2 -611.202} C_VEL
LIN {X 0,Y 601.328,Z 264.727,A -85,B 0,C 180,E1 -612.31,E2 -612.31} C_VEL
LIN {X 0,Y 601.323,Z 267.923,A -85,B 0,C 180,E1 -613.413,E2 -613.413} C_VEL
LIN {X 0,Y 601.327,Z 269.811,A -85,B 0,C 180,E1 -614.407,E2 -614.407} C_VEL
LIN {X 0,Y 601.315,Z 270.593,A -85,B 0,C 180,E1 -615.1,E2 -615.1} C_VEL
LIN {X 0,Y 601.353,Z 270.981,A -85,B 0,C 180,E1 -615.937,E2 -615.937} C_VEL
LIN {X 0,Y 601.325,Z 270.434,A -85,B 0,C 180,E1 -617.17,E2 -617.17} C_VEL
LIN {X 0,Y 601.343,Z 269.527,A -85,B 0,C 180,E1 -617.856,E2 -617.856} C_VEL
LIN {X 0,Y 601.335,Z 266.991,A -85,B 0,C 180,E1 -619.035,E2 -619.035} C_VEL
LIN {X 0,Y 601.343,Z 263.021,A -85,B 0,C 180,E1 -620.244,E2 -620.244} C_VEL
LIN {X 0,Y 601.382,Z 258.458,A -85,B 0,C 180,E1 -621.262,E2 -621.262} C_VEL
LIN {X 0,Y 601.381,Z 251.564,A -85,B 0,C 180,E1 -622.446,E2 -622.446} C_VEL
LIN {X 0,Y 601.378,Z 244.63,A -85,B 0,C 180,E1 -623.394,E2 -623.394} C_VEL
LIN {X 0,Y 601.428,Z 236.548,A -85,B 0,C 180,E1 -624.3,E2 -624.3} C_VEL
LIN {X 0,Y 601.442,Z 227.416,A -85,B 0,C 180,E1 -625.14,E2 -625.14} C_VEL
LIN {X 0,Y 601.499,Z 217.292,A -85,B 0,C 180,E1 -625.896,E2 -625.896} C_VEL
LIN {X 0,Y 601.512,Z 206.147,A -85,B 0,C 180,E1 -626.567,E2 -626.567} C_VEL
LIN {X 0,Y 601.554,Z 195.602,A -85,B 0,C 180,E1 -627.07,E2 -627.07} C_VEL
LIN {X 0,Y 601.533,Z 182.942,A -85,B 0,C 180,E1 -627.531,E2 -627.531} C_VEL
LIN {X 0,Y 601.583,Z 170.193,A -85,B 0,C 180,E1 -627.845,E2 -627.845} C_VEL
LIN {X 0,Y 601.61,Z 152.275,A -85,B 0,C 180,E1 -628.096,E2 -628.096} C_VEL
LIN {X 0,Y 601.495,Z 61.703,A -85,B 0,C 180,E1 -629.184,E2 -629.184} C_VEL
LIN {X 0,Y 601.379,Z 60.855,A -85,B 0,C 180,E1 -629.205,E2 -629.205} C_VEL
LIN {X 0,Y 601.442,Z 45.557,A -85,B 0,C 180,E1 -632.009,E2 -632.009} C_VEL
LIN {X 0,Y 601.434,Z 37.564,A -85,B 0,C 180,E1 -633.517,E2 -633.517} C_VEL
LIN {X 0,Y 601.418,Z 37.565,A -85,B 0,C 180,E1 -636.037,E2 -636.037} C_VEL
LIN {X 0,Y 601.418,Z 37.573,A -85,B 0,C 180,E1 -638.738,E2 -638.738} C_VEL
LIN {X 0,Y 601.417,Z 37.564,A -85,B 0,C 180,E1 -641.459,E2 -641.459} C_VEL
LIN {X 0,Y 601.426,Z 37.569,A -85,B 0,C 180,E1 -644.205,E2 -644.205} C_VEL
LIN {X 0,Y 601.418,Z 37.565,A -85,B 0,C 180,E1 -646.986,E2 -646.986} C_VEL
LIN {X 0,Y 601.407,Z 37.569,A -85,B 0,C 180,E1 -649.81,E2 -649.81} C_VEL
LIN {X 0,Y 601.417,Z 37.566,A -85,B 0,C 180,E1 -652.683,E2 -652.683} C_VEL
LIN {X 0,Y 601.403,Z 37.566,A -85,B 0,C 180,E1 -654.879,E2 -654.879} C_VEL
LIN {X 0,Y 601.421,Z 37.565,A -85,B 0,C 180,E1 -657.362,E2 -657.362} C_VEL
LIN {X 0,Y 601.434,Z 37.568,A -85,B 0,C 180,E1 -660.164,E2 -660.164} C_VEL
LIN {X 0,Y 601.416,Z 37.564,A -85,B 0,C 180,E1 -662.714,E2 -662.714} C_VEL
LIN {X 0,Y 601.42,Z 37.566,A -85,B 0,C 180,E1 -665.114,E2 -665.114} C_VEL
LIN {X 0,Y 601.437,Z 37.568,A -85,B 0,C 180,E1 -667.419,E2 -667.419} C_VEL
LIN {X 0,Y 601.406,Z 37.569,A -85,B 0,C 180,E1 -669.996,E2 -669.996} C_VEL
LIN {X 0,Y 601.412,Z 37.565,A -85,B 0,C 180,E1 -672.67,E2 -672.67} C_VEL
LIN {X 0,Y 601.403,Z 37.574,A -85,B 0,C 180,E1 -675.479,E2 -675.479} C_VEL
LIN {X 0,Y 601.424,Z 37.564,A -85,B 0,C 180,E1 -678.407,E2 -678.407} C_VEL
LIN {X 0,Y 601.433,Z 37.568,A -85,B 0,C 180,E1 -680.875,E2 -680.875} C_VEL
LIN {X 0,Y 601.404,Z 37.57,A -85,B 0,C 180,E1 -683.417,E2 -683.417} C_VEL
LIN {X 0,Y 601.435,Z 37.562,A -85,B 0,C 180,E1 -686.064,E2 -686.064} C_VEL
LIN {X 0,Y 601.416,Z 37.571,A -85,B 0,C 180,E1 -689.057,E2 -689.057} C_VEL
LIN {X 0,Y 601.423,Z 37.565,A -85,B 0,C 180,E1 -691.372,E2 -691.372} C_VEL
LIN {X 0,Y 601.399,Z 37.567,A -85,B 0,C 180,E1 -693.636,E2 -693.636} C_VEL
LIN {X 0,Y 601.419,Z 37.574,A -85,B 0,C 180,E1 -696.589,E2 -696.589} C_VEL
LIN {X 0,Y 601.428,Z 37.563,A -85,B 0,C 180,E1 -699.478,E2 -699.478} C_VEL
LIN {X 0,Y 601.392,Z 37.576,A -85,B 0,C 180,E1 -702.311,E2 -702.311} C_VEL
LIN {X 0,Y 601.409,Z 37.574,A -85,B 0,C 180,E1 -704.408,E2 -704.408} C_VEL
LIN {X 0,Y 601.417,Z 37.564,A -85,B 0,C 180,E1 -707.172,E2 -707.172} C_VEL
LIN {X 0,Y 601.441,Z 37.567,A -85,B 0,C 180,E1 -709.905,E2 -709.905} C_VEL
LIN {X 0,Y 601.407,Z 37.567,A -85,B 0,C 180,E1 -712.614,E2 -712.614} C_VEL
LIN {X 0,Y 601.423,Z 37.565,A -85,B 0,C 180,E1 -715.308,E2 -715.308} C_VEL
LIN {X 0,Y 601.424,Z 37.571,A -85,B 0,C 180,E1 -717.991,E2 -717.991} C_VEL
LIN {X 0,Y 601.443,Z 37.561,A -85,B 0,C 180,E1 -720.669,E2 -720.669} C_VEL
LIN {X 0,Y 601.429,Z 37.568,A -85,B 0,C 180,E1 -723.349,E2 -723.349} C_VEL
LIN {X 0,Y 601.401,Z 37.569,A -85,B 0,C 180,E1 -726.037,E2 -726.037} C_VEL
LIN {X 0,Y 601.434,Z 37.564,A -85,B 0,C 180,E1 -728.061,E2 -728.061} C_VEL
LIN {X 0,Y 601.429,Z 37.567,A -85,B 0,C 180,E1 -731.013,E2 -731.013} C_VEL
LIN {X 0,Y 601.414,Z 37.571,A -85,B 0,C 180,E1 -733.516,E2 -733.516} C_VEL
LIN {X 0,Y 601.435,Z 37.562,A -85,B 0,C 180,E1 -736.287,E2 -736.287} C_VEL
LIN {X 0,Y 601.418,Z 37.574,A -85,B 0,C 180,E1 -739.099,E2 -739.099} C_VEL
LIN {X 0,Y 601.403,Z 37.573,A -85,B 0,C 180,E1 -741.239,E2 -741.239} C_VEL
LIN {X 0,Y 601.457,Z 37.56,A -85,B 0,C 180,E1 -744.14,E2 -744.14} C_VEL
LIN {X 0,Y 601.429,Z 37.568,A -85,B 0,C 180,E1 -747.112,E2 -747.112} C_VEL
LIN {X 0,Y 601.416,Z 37.566,A -85,B 0,C 180,E1 -749.393,E2 -749.393} C_VEL
LIN {X 0,Y 601.401,Z 37.566,A -85,B 0,C 180,E1 -751.727,E2 -751.727} C_VEL
LIN {X 0,Y 601.422,Z 37.566,A -85,B 0,C 180,E1 -754.119,E2 -754.119} C_VEL
LIN {X 0,Y 601.4,Z 37.575,A -85,B 0,C 180,E1 -756.583,E2 -756.583} C_VEL
LIN {X 0,Y 601.406,Z 37.566,A -85,B 0,C 180,E1 -759.127,E2 -759.127} C_VEL
LIN {X 0,Y 601.423,Z 37.566,A -85,B 0,C 180,E1 -761.765,E2 -761.765} C_VEL
LIN {X 0,Y 601.399,Z 37.571,A -85,B 0,C 180,E1 -764.532,E2 -764.532} C_VEL
LIN {X 0,Y 601.412,Z 37.566,A -85,B 0,C 180,E1 -767.409,E2 -767.409} C_VEL
LIN {X 0,Y 601.402,Z 37.576,A -85,B 0,C 180,E1 -770.004,E2 -770.004} C_VEL
LIN {X 0,Y 601.434,Z 37.563,A -85,B 0,C 180,E1 -772.618,E2 -772.618} C_VEL
LIN {X 0,Y 601.417,Z 37.565,A -85,B 0,C 180,E1 -775.068,E2 -775.068} C_VEL
LIN {X 0,Y 601.434,Z 37.567,A -85,B 0,C 180,E1 -777.484,E2 -777.484} C_VEL
LIN {X 0,Y 601.408,Z 37.573,A -85,B 0,C 180,E1 -779.855,E2 -779.855} C_VEL
LIN {X 0,Y 601.402,Z 37.569,A -85,B 0,C 180,E1 -782.131,E2 -782.131} C_VEL
LIN {X 0,Y 601.403,Z 37.567,A -85,B 0,C 180,E1 -784.381,E2 -784.381} C_VEL
LIN {X 0,Y 601.435,Z 37.736,A -85,B 0,C 180,E1 -786.385,E2 -786.385} C_VEL
LIN {X 0,Y 601.73,Z 42.012,A -85,B 0,C 180,E1 -786.966,E2 -786.966} C_VEL
LIN {X 0,Y 601.596,Z 63.848,A -85,B 0,C 180,E1 -789.841,E2 -789.841} C_VEL
LIN {X 0,Y 601.556,Z 85.684,A -85,B 0,C 180,E1 -792.667,E2 -792.667} C_VEL
LIN {X 0,Y 601.451,Z 107.52,A -85,B 0,C 180,E1 -795.45,E2 -795.45} C_VEL
LIN {X 0,Y 601.432,Z 118.353,A -85,B 0,C 180,E1 -796.818,E2 -796.818} C_VEL
LIN {X 0,Y 601.631,Z 138.8,A -85,B 0,C 180,E1 -797.069,E2 -797.069} C_VEL
LIN {X 0,Y 601.595,Z 226.935,A -85,B 0,C 180,E1 -798.139,E2 -798.139} C_VEL
LIN {X 0,Y 601.581,Z 240.21,A -85,B 0,C 180,E1 -798.438,E2 -798.438} C_VEL
LIN {X 0,Y 601.547,Z 251.894,A -85,B 0,C 180,E1 -798.825,E2 -798.825} C_VEL
LIN {X 0,Y 601.522,Z 264.629,A -85,B 0,C 180,E1 -799.396,E2 -799.396} C_VEL
LIN {X 0,Y 601.475,Z 276.196,A -85,B 0,C 180,E1 -800.075,E2 -800.075} C_VEL
LIN {X 0,Y 601.444,Z 286.593,A -85,B 0,C 180,E1 -800.839,E2 -800.839} C_VEL
LIN {X 0,Y 601.429,Z 295.11,A -85,B 0,C 180,E1 -801.601,E2 -801.601} C_VEL
LIN {X 0,Y 601.418,Z 302.958,A -85,B 0,C 180,E1 -802.446,E2 -802.446} C_VEL
LIN {X 0,Y 601.37,Z 310.224,A -85,B 0,C 180,E1 -803.398,E2 -803.398} C_VEL
LIN {X 0,Y 601.372,Z 315.865,A -85,B 0,C 180,E1 -804.299,E2 -804.299} C_VEL
LIN {X 0,Y 601.336,Z 320.949,A -85,B 0,C 180,E1 -805.307,E2 -805.307} C_VEL
LIN {X 0,Y 601.368,Z 324.895,A -85,B 0,C 180,E1 -806.314,E2 -806.314} C_VEL
LIN {X 0,Y 601.325,Z 327.808,A -85,B 0,C 180,E1 -807.32,E2 -807.32} C_VEL
LIN {X 0,Y 601.343,Z 329.201,A -85,B 0,C 180,E1 -807.99,E2 -807.99} C_VEL
LIN {X 0,Y 601.339,Z 330.784,A -85,B 0,C 180,E1 -809.33,E2 -809.33} C_VEL
LIN {X 0,Y 601.335,Z 331,A -85,B 0,C 180,E1 -810,E2 -810} C_VEL
LIN {X 0,Y 601.347,Z 330.185,A -85,B 0,C 180,E1 -811.339,E2 -811.339} C_VEL
LIN {X 0,Y 601.343,Z 329.202,A -85,B 0,C 180,E1 -812.009,E2 -812.009} C_VEL
LIN {X 0,Y 601.325,Z 327.81,A -85,B 0,C 180,E1 -812.679,E2 -812.679} C_VEL
LIN {X 0,Y 601.368,Z 324.897,A -85,B 0,C 180,E1 -813.685,E2 -813.685} C_VEL
LIN {X 0,Y 601.336,Z 320.951,A -85,B 0,C 180,E1 -814.692,E2 -814.692} C_VEL
LIN {X 0,Y 601.372,Z 314.879,A -85,B 0,C 180,E1 -815.869,E2 -815.869} C_VEL
LIN {X 0,Y 601.381,Z 308.238,A -85,B 0,C 180,E1 -816.879,E2 -816.879} C_VEL
LIN {X 0,Y 601.4,Z 299.992,A -85,B 0,C 180,E1 -817.892,E2 -817.892} C_VEL
LIN {X 0,Y 601.436,Z 291.54,A -85,B 0,C 180,E1 -818.737,E2 -818.737} C_VEL
LIN {X 0,Y 601.447,Z 281.097,A -85,B 0,C 180,E1 -819.585,E2 -819.585} C_VEL
LIN {X 0,Y 601.463,Z 270.763,A -85,B 0,C 180,E1 -820.264,E2 -820.264} C_VEL
LIN {X 0,Y 601.538,Z 258.591,A -85,B 0,C 180,E1 -820.896,E2 -820.896} C_VEL
LIN {X 0,Y 601.563,Z 246.223,A -85,B 0,C 180,E1 -821.378,E2 -821.378} C_VEL
LIN {X 0,Y 601.583,Z 233.449,A -85,B 0,C 180,E1 -821.733,E2 -821.733} C_VEL
LIN {X 0,Y 601.622,Z 221.105,A -85,B 0,C 180,E1 -821.945,E2 -821.945} C_VEL
LIN {X 0,Y 601.542,Z 119.165,A -85,B 0,C 180,E1 -823.169,E2 -823.169} C_VEL
LIN {X 0,Y 601.438,Z 118.272,A -85,B 0,C 180,E1 -823.193,E2 -823.193} C_VEL
LIN {X 0,Y 601.503,Z 95.242,A -85,B 0,C 180,E1 -826.111,E2 -826.111} C_VEL
LIN {X 0,Y 601.583,Z 75.684,A -85,B 0,C 180,E1 -828.621,E2 -828.621} C_VEL
LIN {X 0,Y 601.659,Z 54.299,A -85,B 0,C 180,E1 -831.409,E2 -831.409} C_VEL
LIN {X 0,Y 601.74,Z 39.287,A -85,B 0,C 180,E1 -833.397,E2 -833.397} C_VEL
LIN {X 0,Y 601.417,Z 37.568,A -85,B 0,C 180,E1 -833.638,E2 -833.638} C_VEL
LIN {X 0,Y 601.403,Z 37.576,A -85,B 0,C 180,E1 -836.363,E2 -836.363} C_VEL
LIN {X 0,Y 601.44,Z 37.565,A -85,B 0,C 180,E1 -838.789,E2 -838.789} C_VEL
LIN {X 0,Y 601.418,Z 37.565,A -85,B 0,C 180,E1 -841.454,E2 -841.454} C_VEL
LIN {X 0,Y 601.422,Z 37.574,A -85,B 0,C 180,E1 -844.118,E2 -844.118} C_VEL
LIN {X 0,Y 601.41,Z 37.567,A -85,B 0,C 180,E1 -846.582,E2 -846.582} C_VEL
LIN {X 0,Y 601.41,Z 37.566,A -85,B 0,C 180,E1 -849.126,E2 -849.126} C_VEL
LIN {X 0,Y 601.422,Z 37.574,A -85,B 0,C 180,E1 -851.765,E2 -851.765} C_VEL
LIN {X 0,Y 601.396,Z 37.567,A -85,B 0,C 180,E1 -854.532,E2 -854.532} C_VEL
LIN {X 0,Y 601.412,Z 37.573,A -85,B 0,C 180,E1 -857.409,E2 -857.409} C_VEL
LIN {X 0,Y 601.439,Z 37.562,A -85,B 0,C 180,E1 -860.464,E2 -860.464} C_VEL
LIN {X 0,Y 601.409,Z 37.573,A -85,B 0,C 180,E1 -863.417,E2 -863.417} C_VEL
LIN {X 0,Y 601.431,Z 37.563,A -85,B 0,C 180,E1 -866.064,E2 -866.064} C_VEL
LIN {X 0,Y 601.428,Z 37.565,A -85,B 0,C 180,E1 -868.543,E2 -868.543} C_VEL
LIN {X 0,Y 601.427,Z 37.567,A -85,B 0,C 180,E1 -871.373,E2 -871.373} C_VEL
LIN {X 0,Y 601.401,Z 37.567,A -85,B 0,C 180,E1 -873.636,E2 -873.636} C_VEL
LIN {X 0,Y 601.417,Z 37.572,A -85,B 0,C 180,E1 -876.59,E2 -876.59} C_VEL
LIN {X 0,Y 601.427,Z 37.563,A -85,B 0,C 180,E1 -879.478,E2 -879.478} C_VEL
LIN {X 0,Y 601.394,Z 37.574,A -85,B 0,C 180,E1 -882.312,E2 -882.312} C_VEL
LIN {X 0,Y 601.41,Z 37.575,A -85,B 0,C 180,E1 -884.409,E2 -884.409} C_VEL
LIN {X 0,Y 601.417,Z 37.564,A -85,B 0,C 180,E1 -887.172,E2 -887.172} C_VEL
LIN {X 0,Y 601.441,Z 37.567,A -85,B 0,C 180,E1 -889.905,E2 -889.905} C_VEL
LIN {X 0,Y 601.405,Z 37.567,A -85,B 0,C 180,E1 -892.615,E2 -892.615} C_VEL
LIN {X 0,Y 601.423,Z 37.565,A -85,B 0,C 180,E1 -895.308,E2 -895.308} C_VEL
LIN {X 0,Y 601.421,Z 37.571,A -85,B 0,C 180,E1 -897.991,E2 -897.991} C_VEL
LIN {X 0,Y 601.441,Z 37.561,A -85,B 0,C 180,E1 -900.67,E2 -900.67} C_VEL
LIN {X 0,Y 601.429,Z 37.568,A -85,B 0,C 180,E1 -903.35,E2 -903.35} C_VEL
LIN {X 0,Y 601.395,Z 37.569,A -85,B 0,C 180,E1 -906.037,E2 -906.037} C_VEL
LIN {X 0,Y 601.415,Z 37.566,A -85,B 0,C 180,E1 -908.738,E2 -908.738} C_VEL
LIN {X 0,Y 601.432,Z 37.569,A -85,B 0,C 180,E1 -911.458,E2 -911.458} C_VEL
LIN {X 0,Y 601.402,Z 37.566,A -85,B 0,C 180,E1 -912.369,E2 -912.369} C_VEL
LIN {X 0,Y 600.746,Z 37.655,A -85,B 0,C 180,E1 -912.928,E2 -912.928} C_VEL
LIN {X 0,Y 597.9,Z 38.013,A -85,B 0,C 180,E1 -913.836,E2 -913.836} C_VEL
LIN {X 0,Y 595.487,Z 38.315,A -85,B 0,C 180,E1 -914.566,E2 -914.566} C_VEL
LIN {X 0,Y 594.444,Z 38.443,A -85,B 0,C 180,E1 -915.13,E2 -915.13} C_VEL
LIN {X 0,Y 594.356,Z 38.449,A -85,B 0,C 180,E1 -915.32,E2 -915.32} C_VEL
LIN {X 0,Y 594.384,Z 38.447,A -85,B 0,C 180,E1 -917.194,E2 -917.194} C_VEL
LIN {X 0,Y 594.369,Z 38.443,A -85,B 0,C 180,E1 -920.054,E2 -920.054} C_VEL
LIN {X 0,Y 594.353,Z 38.451,A -85,B 0,C 180,E1 -922.968,E2 -922.968} C_VEL
LIN {X 0,Y 594.355,Z 38.446,A -85,B 0,C 180,E1 -925.194,E2 -925.194} C_VEL
LIN {X 0,Y 594.34,Z 38.446,A -85,B 0,C 180,E1 -927.519,E2 -927.519} C_VEL
LIN {X 0,Y 594.384,Z 38.448,A -85,B 0,C 180,E1 -930.328,E2 -930.328} C_VEL
LIN {X 0,Y 594.375,Z 38.443,A -85,B 0,C 180,E1 -932.951,E2 -932.951} C_VEL
LIN {X 0,Y 594.324,Z 38.448,A -85,B 0,C 180,E1 -935.411,E2 -935.411} C_VEL
LIN {X 0,Y 594.383,Z 38.447,A -85,B 0,C 180,E1 -937.941,E2 -937.941} C_VEL
LIN {X 0,Y 594.362,Z 38.443,A -85,B 0,C 180,E1 -940.821,E2 -940.821} C_VEL
LIN {X 0,Y 594.342,Z 38.448,A -85,B 0,C 180,E1 -943.302,E2 -943.302} C_VEL
LIN {X 0,Y 594.343,Z 38.45,A -85,B 0,C 180,E1 -946.164,E2 -946.164} C_VEL
LIN {X 0,Y 594.362,Z 38.444,A -85,B 0,C 180,E1 -948.535,E2 -948.535} C_VEL
LIN {X 0,Y 594.364,Z 38.449,A -85,B 0,C 180,E1 -951.299,E2 -951.299} C_VEL
LIN {X 0,Y 594.344,Z 38.451,A -85,B 0,C 180,E1 -953.755,E2 -953.755} C_VEL
LIN {X 0,Y 594.344,Z 38.447,A -85,B 0,C 180,E1 -956.237,E2 -956.237} C_VEL
LIN {X 0,Y 594.365,Z 38.588,A -85,B 0,C 180,E1 -958.578,E2 -958.578} C_VEL
LIN {X 0,Y 594.388,Z 51.758,A -85,B 0,C 180,E1 -961.042,E2 -961.042} C_VEL
LIN {X 0,Y 594.353,Z 60.869,A -85,B 0,C 180,E1 -962.729,E2 -962.729} C_VEL
LIN {X 0,Y 594.771,Z 66.218,A -85,B 0,C 180,E1 -962.809,E2 -962.809} C_VEL
LIN {X 0,Y 594.682,Z 167.05,A -85,B 0,C 180,E1 -964.046,E2 -964.046} C_VEL
LIN {X 0,Y 594.64,Z 180.374,A -85,B 0,C 180,E1 -964.351,E2 -964.351} C_VEL
LIN {X 0,Y 594.552,Z 192.719,A -85,B 0,C 180,E1 -964.768,E2 -964.768} C_VEL
LIN {X 0,Y 594.498,Z 204.159,A -85,B 0,C 180,E1 -965.289,E2 -965.289} C_VEL
LIN {X 0,Y 594.415,Z 215.085,A -85,B 0,C 180,E1 -965.927,E2 -965.927} C_VEL
LIN {X 0,Y 594.422,Z 226.407,A -85,B 0,C 180,E1 -966.759,E2 -966.759} C_VEL
LIN {X 0,Y 594.373,Z 235.884,A -85,B 0,C 180,E1 -967.622,E2 -967.622} C_VEL
LIN {X 0,Y 594.343,Z 245.095,A -85,B 0,C 180,E1 -968.667,E2 -968.667} C_VEL
LIN {X 0,Y 594.302,Z 252.84,A -85,B 0,C 180,E1 -969.764,E2 -969.764} C_VEL
LIN {X 0,Y 594.248,Z 259.205,A -85,B 0,C 180,E1 -970.923,E2 -970.923} C_VEL
LIN {X 0,Y 594.241,Z 264.099,A -85,B 0,C 180,E1 -972.092,E2 -972.092} C_VEL
LIN {X 0,Y 594.239,Z 267.808,A -85,B 0,C 180,E1 -973.333,E2 -973.333} C_VEL
LIN {X 0,Y 594.225,Z 269.534,A -85,B 0,C 180,E1 -974.216,E2 -974.216} C_VEL
LIN {X 0,Y 594.211,Z 270.448,A -85,B 0,C 180,E1 -974.918,E2 -974.918} C_VEL
LIN {X 0,Y 594.264,Z 270.967,A -85,B 0,C 180,E1 -975.877,E2 -975.877} C_VEL
LIN {X 0,Y 594.244,Z 270.582,A -85,B 0,C 180,E1 -977.015,E2 -977.015} C_VEL
LIN {X 0,Y 594.24,Z 269.801,A -85,B 0,C 180,E1 -977.709,E2 -977.709} C_VEL
LIN {X 0,Y 594.252,Z 267.182,A -85,B 0,C 180,E1 -978.998,E2 -978.998} C_VEL
LIN {X 0,Y 594.258,Z 263.633,A -85,B 0,C 180,E1 -980.126,E2 -980.126} C_VEL
LIN {X 0,Y 594.293,Z 259.254,A -85,B 0,C 180,E1 -981.157,E2 -981.157} C_VEL
LIN {X 0,Y 594.3,Z 253.692,A -85,B 0,C 180,E1 -982.184,E2 -982.184} C_VEL
LIN {X 0,Y 594.32,Z 246.772,A -85,B 0,C 180,E1 -983.209,E2 -983.209} C_VEL
LIN {X 0,Y 594.345,Z 238.137,A -85,B 0,C 180,E1 -984.232,E2 -984.232} C_VEL
LIN {X 0,Y 594.417,Z 229.32,A -85,B 0,C 180,E1 -985.083,E2 -985.083} C_VEL
LIN {X 0,Y 594.458,Z 218.506,A -85,B 0,C 180,E1 -985.933,E2 -985.933} C_VEL
LIN {X 0,Y 594.529,Z 207.615,A -85,B 0,C 180,E1 -986.612,E2 -986.612} C_VEL
LIN {X 0,Y 594.562,Z 195.514,A -85,B 0,C 180,E1 -987.205,E2 -987.205} C_VEL
LIN {X 0,Y 594.587,Z 182.79,A -85,B 0,C 180,E1 -987.672,E2 -987.672} C_VEL
LIN {X 0,Y 594.656,Z 169.938,A -85,B 0,C 180,E1 -987.99,E2 -987.99} C_VEL
LIN {X 0,Y 594.671,Z 151.914,A -85,B 0,C 180,E1 -988.244,E2 -988.244} C_VEL
LIN {X 0,Y 594.66,Z 62.937,A -85,B 0,C 180,E1 -989.323,E2 -989.323} C_VEL
LIN {X 0,Y 594.329,Z 60.85,A -85,B 0,C 180,E1 -989.365,E2 -989.365} C_VEL
LIN {X 0,Y 594.411,Z 46.468,A -85,B 0,C 180,E1 -992.033,E2 -992.033} C_VEL
LIN {X 0,Y 594.408,Z 38.44,A -85,B 0,C 180,E1 -993.559,E2 -993.559} C_VEL
LIN {X 0,Y 594.406,Z 38.448,A -85,B 0,C 180,E1 -996.691,E2 -996.691} C_VEL
LIN {X 0,Y 594.384,Z 38.447,A -85,B 0,C 180,E1 -998.842,E2 -998.842} C_VEL
LIN {X 0,Y 594.385,Z 38.44,A -85,B 0,C 180,E1 -1001.596,E2 -1001.596} C_VEL
LIN {X 0,Y 594.396,Z 38.448,A -85,B 0,C 180,E1 -1004.377,E2 -1004.377} C_VEL
LIN {X 0,Y 594.383,Z 38.441,A -85,B 0,C 180,E1 -1007.194,E2 -1007.194} C_VEL
LIN {X 0,Y 594.375,Z 38.448,A -85,B 0,C 180,E1 -1010.054,E2 -1010.054} C_VEL
LIN {X 0,Y 594.362,Z 38.443,A -85,B 0,C 180,E1 -1012.968,E2 -1012.968} C_VEL
LIN {X 0,Y 594.376,Z 38.441,A -85,B 0,C 180,E1 -1015.193,E2 -1015.193} C_VEL
LIN {X 0,Y 594.392,Z 38.442,A -85,B 0,C 180,E1 -1017.527,E2 -1017.527} C_VEL
LIN {X 0,Y 594.391,Z 38.443,A -85,B 0,C 180,E1 -1020.328,E2 -1020.328} C_VEL
LIN {X 0,Y 594.38,Z 38.441,A -85,B 0,C 180,E1 -1022.95,E2 -1022.95} C_VEL
LIN {X 0,Y 594.362,Z 38.448,A -85,B 0,C 180,E1 -1025.408,E2 -1025.408} C_VEL
LIN {X 0,Y 594.383,Z 38.445,A -85,B 0,C 180,E1 -1027.941,E2 -1027.941} C_VEL
LIN {X 0,Y 594.377,Z 38.442,A -85,B 0,C 180,E1 -1030.821,E2 -1030.821} C_VEL
LIN {X 0,Y 594.37,Z 38.45,A -85,B 0,C 180,E1 -1033.299,E2 -1033.299} C_VEL
LIN {X 0,Y 594.364,Z 38.443,A -85,B 0,C 180,E1 -1036.161,E2 -1036.161} C_VEL
LIN {X 0,Y 594.381,Z 38.441,A -85,B 0,C 180,E1 -1038.536,E2 -1038.536} C_VEL
LIN {X 0,Y 594.382,Z 38.448,A -85,B 0,C 180,E1 -1041.296,E2 -1041.296} C_VEL
LIN {X 0,Y 594.354,Z 38.445,A -85,B 0,C 180,E1 -1043.755,E2 -1043.755} C_VEL
LIN {X 0,Y 594.378,Z 38.442,A -85,B 0,C 180,E1 -1046.238,E2 -1046.238} C_VEL
LIN {X 0,Y 594.373,Z 38.448,A -85,B 0,C 180,E1 -1048.65,E2 -1048.65} C_VEL
LIN {X 0,Y 594.384,Z 38.446,A -85,B 0,C 180,E1 -1051.042,E2 -1051.042} C_VEL
LIN {X 0,Y 594.383,Z 38.442,A -85,B 0,C 180,E1 -1053.3,E2 -1053.3} C_VEL
LIN {X 0,Y 594.391,Z 38.444,A -85,B 0,C 180,E1 -1056.296,E2 -1056.296} C_VEL
LIN {X 0,Y 594.401,Z 38.439,A -85,B 0,C 180,E1 -1059.224,E2 -1059.224} C_VEL
LIN {X 0,Y 594.351,Z 38.449,A -85,B 0,C 180,E1 -1062.095,E2 -1062.095} C_VEL
LIN {X 0,Y 594.364,Z 38.451,A -85,B 0,C 180,E1 -1064.219,E2 -1064.219} C_VEL
LIN {X 0,Y 594.38,Z 38.45,A -85,B 0,C 180,E1 -1066.321,E2 -1066.321} C_VEL
LIN {X 0,Y 594.377,Z 38.441,A -85,B 0,C 180,E1 -1069.094,E2 -1069.094} C_VEL
LIN {X 0,Y 594.416,Z 38.443,A -85,B 0,C 180,E1 -1071.843,E2 -1071.843} C_VEL
LIN {X 0,Y 594.385,Z 38.442,A -85,B 0,C 180,E1 -1074.572,E2 -1074.572} C_VEL
LIN {X 0,Y 594.408,Z 38.439,A -85,B 0,C 180,E1 -1077.289,E2 -1077.289} C_VEL
LIN {X 0,Y 594.412,Z 38.443,A -85,B 0,C 180,E1 -1080,E2 -1080} C_VEL
LIN {X 0,Y 594.403,Z 38.438,A -85,B 0,C 180,E1 -1082.711,E2 -1082.711} C_VEL
LIN {X 0,Y 594.39,Z 38.447,A -85,B 0,C 180,E1 -1085.428,E2 -1085.428} C_VEL
LIN {X 0,Y 594.381,Z 38.442,A -85,B 0,C 180,E1 -1088.157,E2 -1088.157} C_VEL
LIN {X 0,Y 594.393,Z 38.444,A -85,B 0,C 180,E1 -1091.074,E2 -1091.074} C_VEL
LIN {X 0,Y 594.375,Z 38.446,A -85,B 0,C 180,E1 -1093.679,E2 -1093.679} C_VEL
LIN {X 0,Y 594.396,Z 38.442,A -85,B 0,C 180,E1 -1096.719,E2 -1096.719} C_VEL
LIN {X 0,Y 594.367,Z 38.449,A -85,B 0,C 180,E1 -1099.334,E2 -1099.334} C_VEL
LIN {X 0,Y 594.364,Z 38.446,A -85,B 0,C 180,E1 -1101.503,E2 -1101.503} C_VEL
LIN {X 0,Y 594.391,Z 38.442,A -85,B 0,C 180,E1 -1104.446,E2 -1104.446} C_VEL
LIN {X 0,Y 594.377,Z 38.443,A -85,B 0,C 180,E1 -1107.461,E2 -1107.461} C_VEL
LIN {X 0,Y 594.387,Z 38.444,A -85,B 0,C 180,E1 -1110.328,E2 -1110.328} C_VEL
LIN {X 0,Y 594.378,Z 38.446,A -85,B 0,C 180,E1 -1112.95,E2 -1112.95} C_VEL
LIN {X 0,Y 594.353,Z 38.444,A -85,B 0,C 180,E1 -1115.409,E2 -1115.409} C_VEL
LIN {X 0,Y 594.386,Z 38.442,A -85,B 0,C 180,E1 -1117.941,E2 -1117.941} C_VEL
LIN {X 0,Y 594.372,Z 38.445,A -85,B 0,C 180,E1 -1120.821,E2 -1120.821} C_VEL
LIN {X 0,Y 594.367,Z 38.442,A -85,B 0,C 180,E1 -1123.3,E2 -1123.3} C_VEL
LIN {X 0,Y 594.362,Z 38.453,A -85,B 0,C 180,E1 -1126.161,E2 -1126.161} C_VEL
LIN {X 0,Y 594.375,Z 38.445,A -85,B 0,C 180,E1 -1128.535,E2 -1128.535} C_VEL
LIN {X 0,Y 594.374,Z 38.443,A -85,B 0,C 180,E1 -1131.297,E2 -1131.297} C_VEL
LIN {X 0,Y 594.353,Z 38.452,A -85,B 0,C 180,E1 -1133.755,E2 -1133.755} C_VEL
LIN {X 0,Y 594.367,Z 38.446,A -85,B 0,C 180,E1 -1136.238,E2 -1136.238} C_VEL
LIN {X 0,Y 594.369,Z 38.442,A -85,B 0,C 180,E1 -1138.649,E2 -1138.649} C_VEL
LIN {X 0,Y 594.386,Z 38.443,A -85,B 0,C 180,E1 -1141.042,E2 -1141.042} C_VEL
LIN {X 0,Y 594.377,Z 38.446,A -85,B 0,C 180,E1 -1143.98,E2 -1143.98} C_VEL
LIN {X 0,Y 594.405,Z 38.604,A -85,B 0,C 180,E1 -1146.25,E2 -1146.25} C_VEL
LIN {X 0,Y 594.812,Z 43.171,A -85,B 0,C 180,E1 -1146.867,E2 -1146.867} C_VEL
LIN {X 0,Y 594.693,Z 63.848,A -85,B 0,C 180,E1 -1149.596,E2 -1149.596} C_VEL
LIN {X 0,Y 594.598,Z 85.684,A -85,B 0,C 180,E1 -1152.458,E2 -1152.458} C_VEL
LIN {X 0,Y 594.443,Z 107.52,A -85,B 0,C 180,E1 -1155.274,E2 -1155.274} C_VEL
LIN {X 0,Y 594.435,Z 118.353,A -85,B 0,C 180,E1 -1156.66,E2 -1156.66} C_VEL
LIN {X 0,Y 594.741,Z 124.49,A -85,B 0,C 180,E1 -1156.743,E2 -1156.743} C_VEL
LIN {X 0,Y 594.664,Z 226.935,A -85,B 0,C 180,E1 -1157.999,E2 -1157.999} C_VEL
LIN {X 0,Y 594.624,Z 240.211,A -85,B 0,C 180,E1 -1158.301,E2 -1158.301} C_VEL
LIN {X 0,Y 594.592,Z 253.265,A -85,B 0,C 180,E1 -1158.745,E2 -1158.745} C_VEL
LIN {X 0,Y 594.536,Z 264.627,A -85,B 0,C 180,E1 -1159.27,E2 -1159.27} C_VEL
LIN {X 0,Y 594.471,Z 276.198,A -85,B 0,C 180,E1 -1159.957,E2 -1159.957} C_VEL
LIN {X 0,Y 594.414,Z 286.595,A -85,B 0,C 180,E1 -1160.729,E2 -1160.729} C_VEL
LIN {X 0,Y 594.383,Z 295.11,A -85,B 0,C 180,E1 -1161.5,E2 -1161.5} C_VEL
LIN {X 0,Y 594.347,Z 302.959,A -85,B 0,C 180,E1 -1162.355,E2 -1162.355} C_VEL
LIN {X 0,Y 594.283,Z 310.812,A -85,B 0,C 180,E1 -1163.408,E2 -1163.408} C_VEL
LIN {X 0,Y 594.289,Z 317.679,A -85,B 0,C 180,E1 -1164.571,E2 -1164.571} C_VEL
LIN {X 0,Y 594.27,Z 322.371,A -85,B 0,C 180,E1 -1165.591,E2 -1165.591} C_VEL
LIN {X 0,Y 594.267,Z 325.956,A -85,B 0,C 180,E1 -1166.61,E2 -1166.61} C_VEL
LIN {X 0,Y 594.226,Z 327.808,A -85,B 0,C 180,E1 -1167.288,E2 -1167.288} C_VEL
LIN {X 0,Y 594.242,Z 329.2,A -85,B 0,C 180,E1 -1167.966,E2 -1167.966} C_VEL
LIN {X 0,Y 594.239,Z 330.784,A -85,B 0,C 180,E1 -1169.322,E2 -1169.322} C_VEL
LIN {X 0,Y 594.236,Z 331,A -85,B 0,C 180,E1 -1170,E2 -1170} C_VEL
LIN {X 0,Y 594.247,Z 330.185,A -85,B 0,C 180,E1 -1171.355,E2 -1171.355} C_VEL
LIN {X 0,Y 594.242,Z 329.201,A -85,B 0,C 180,E1 -1172.033,E2 -1172.033} C_VEL
LIN {X 0,Y 594.226,Z 327.81,A -85,B 0,C 180,E1 -1172.711,E2 -1172.711} C_VEL
LIN {X 0,Y 594.289,Z 324.897,A -85,B 0,C 180,E1 -1173.729,E2 -1173.729} C_VEL
LIN {X 0,Y 594.241,Z 320.95,A -85,B 0,C 180,E1 -1174.749,E2 -1174.749} C_VEL
LIN {X 0,Y 594.305,Z 314.879,A -85,B 0,C 180,E1 -1175.939,E2 -1175.939} C_VEL
LIN {X 0,Y 594.308,Z 308.239,A -85,B 0,C 180,E1 -1176.962,E2 -1176.962} C_VEL
LIN {X 0,Y 594.359,Z 299.992,A -85,B 0,C 180,E1 -1177.986,E2 -1177.986} C_VEL
LIN {X 0,Y 594.382,Z 291.541,A -85,B 0,C 180,E1 -1178.842,E2 -1178.842} C_VEL
LIN {X 0,Y 594.428,Z 281.099,A -85,B 0,C 180,E1 -1179.699,E2 -1179.699} C_VEL
LIN {X 0,Y 594.471,Z 270.762,A -85,B 0,C 180,E1 -1180.386,E2 -1180.386} C_VEL
LIN {X 0,Y 594.558,Z 259.721,A -85,B 0,C 180,E1 -1180.973,E2 -1180.973} C_VEL
LIN {X 0,Y 594.583,Z 247.717,A -85,B 0,C 180,E1 -1181.464,E2 -1181.464} C_VEL
LIN {X 0,Y 594.633,Z 234.362,A -85,B 0,C 180,E1 -1181.85,E2 -1181.85} C_VEL
LIN {X 0,Y 594.694,Z 221.105,A -85,B 0,C 180,E1 -1182.087,E2 -1182.087} C_VEL
LIN {X 0,Y 594.635,Z 119.836,A -85,B 0,C 180,E1 -1183.316,E2 -1183.316} C_VEL
LIN {X 0,Y 594.442,Z 118.272,A -85,B 0,C 180,E1 -1183.351,E2 -1183.351} C_VEL
LIN {X 0,Y 594.524,Z 95.242,A -85,B 0,C 180,E1 -1186.305,E2 -1186.305} C_VEL
LIN {X 0,Y 594.604,Z 75.479,A -85,B 0,C 180,E1 -1188.875,E2 -1188.875} C_VEL
LIN {X 0,Y 594.74,Z 55.664,A -85,B 0,C 180,E1 -1191.489,E2 -1191.489} C_VEL
LIN {X 0,Y 594.728,Z 40.349,A -85,B 0,C 180,E1 -1193.505,E2 -1193.505} C_VEL
LIN {X 0,Y 594.387,Z 38.446,A -85,B 0,C 180,E1 -1193.796,E2 -1193.796} C_VEL
LIN {X 0,Y 594.387,Z 38.446,A -85,B 0,C 180,E1 -1196.699,E2 -1196.699} C_VEL
LIN {X 0,Y 594.381,Z 38.442,A -85,B 0,C 180,E1 -1198.998,E2 -1198.998} C_VEL
LIN {X 0,Y 594.376,Z 38.444,A -85,B 0,C 180,E1 -1201.642,E2 -1201.642} C_VEL
LIN {X 0,Y 594.394,Z 38.442,A -85,B 0,C 180,E1 -1204.579,E2 -1204.579} C_VEL
LIN {X 0,Y 594.383,Z 38.441,A -85,B 0,C 180,E1 -1207.086,E2 -1207.086} C_VEL
LIN {X 0,Y 594.358,Z 38.453,A -85,B 0,C 180,E1 -1209.772,E2 -1209.772} C_VEL
LIN {X 0,Y 594.367,Z 38.444,A -85,B 0,C 180,E1 -1212.375,E2 -1212.375} C_VEL
LIN {X 0,Y 594.354,Z 38.447,A -85,B 0,C 180,E1 -1215.192,E2 -1215.192} C_VEL
LIN {X 0,Y 594.381,Z 38.442,A -85,B 0,C 180,E1 -1218.151,E2 -1218.151} C_VEL
LIN {X 0,Y 594.384,Z 38.448,A -85,B 0,C 180,E1 -1221.195,E2 -1221.195} C_VEL
LIN {X 0,Y 594.394,Z 38.442,A -85,B 0,C 180,E1 -1223.758,E2 -1223.758} C_VEL
LIN {X 0,Y 594.377,Z 38.441,A -85,B 0,C 180,E1 -1226.239,E2 -1226.239} C_VEL
LIN {X 0,Y 594.378,Z 38.445,A -85,B 0,C 180,E1 -1228.65,E2 -1228.65} C_VEL
LIN {X 0,Y 594.381,Z 38.45,A -85,B 0,C 180,E1 -1231.042,E2 -1231.042} C_VEL
LIN {X 0,Y 594.382,Z 38.441,A -85,B 0,C 180,E1 -1233.977,E2 -1233.977} C_VEL
LIN {X 0,Y 594.389,Z 38.443,A -85,B 0,C 180,E1 -1236.296,E2 -1236.296} C_VEL
LIN {X 0,Y 594.4,Z 38.44,A -85,B 0,C 180,E1 -1239.224,E2 -1239.224} C_VEL
LIN {X 0,Y 594.351,Z 38.448,A -85,B 0,C 180,E1 -1242.095,E2 -1242.095} C_VEL
LIN {X 0,Y 594.365,Z 38.45,A -85,B 0,C 180,E1 -1244.219,E2 -1244.219} C_VEL
LIN {X 0,Y 594.377,Z 38.451,A -85,B 0,C 180,E1 -1246.321,E2 -1246.321} C_VEL
LIN {X 0,Y 594.375,Z 38.442,A -85,B 0,C 180,E1 -1249.095,E2 -1249.095} C_VEL
LIN {X 0,Y 594.416,Z 38.442,A -85,B 0,C 180,E1 -1251.843,E2 -1251.843} C_VEL
LIN {X 0,Y 594.384,Z 38.442,A -85,B 0,C 180,E1 -1254.572,E2 -1254.572} C_VEL
LIN {X 0,Y 594.407,Z 38.439,A -85,B 0,C 180,E1 -1257.289,E2 -1257.289} C_VEL
LIN {X 0,Y 594.407,Z 38.443,A -85,B 0,C 180,E1 -1260,E2 -1260} C_VEL
LIN {X 0,Y 594.4,Z 38.438,A -85,B 0,C 180,E1 -1262.711,E2 -1262.711} C_VEL
LIN {X 0,Y 594.39,Z 38.448,A -85,B 0,C 180,E1 -1265.428,E2 -1265.428} C_VEL
LIN {X 0,Y 594.36,Z 38.444,A -85,B 0,C 180,E1 -1268.158,E2 -1268.158} C_VEL
LIN {X 0,Y 594.391,Z 38.446,A -85,B 0,C 180,E1 -1271.076,E2 -1271.076} C_VEL
LIN {X 0,Y 594.369,Z 38.445,A -85,B 0,C 180,E1 -1273.679,E2 -1273.679} C_VEL
LIN {X 0,Y 594.356,Z 38.449,A -85,B 0,C 180,E1 -1275.32,E2 -1275.32} C_VEL
LIN {X 0,Y 593.677,Z 38.531,A -85,B 0,C 180,E1 -1275.886,E2 -1275.886} C_VEL
LIN {X 0,Y 590.805,Z 38.893,A -85,B 0,C 180,E1 -1276.804,E2 -1276.804} C_VEL
LIN {X 0,Y 588.394,Z 39.189,A -85,B 0,C 180,E1 -1277.543,E2 -1277.543} C_VEL
LIN {X 0,Y 587.375,Z 39.313,A -85,B 0,C 180,E1 -1278.113,E2 -1278.113} C_VEL
LIN {X 0,Y 587.3,Z 39.324,A -85,B 0,C 180,E1 -1278.306,E2 -1278.306} C_VEL
LIN {X 0,Y 587.329,Z 39.325,A -85,B 0,C 180,E1 -1281.038,E2 -1281.038} C_VEL
LIN {X 0,Y 587.31,Z 39.324,A -85,B 0,C 180,E1 -1283.26,E2 -1283.26} C_VEL
LIN {X 0,Y 587.318,Z 39.32,A -85,B 0,C 180,E1 -1285.518,E2 -1285.518} C_VEL
LIN {X 0,Y 587.303,Z 39.323,A -85,B 0,C 180,E1 -1287.82,E2 -1287.82} C_VEL
LIN {X 0,Y 587.332,Z 39.328,A -85,B 0,C 180,E1 -1290.51,E2 -1290.51} C_VEL
LIN {X 0,Y 587.325,Z 39.32,A -85,B 0,C 180,E1 -1293.398,E2 -1293.398} C_VEL
LIN {X 0,Y 587.285,Z 39.329,A -85,B 0,C 180,E1 -1295.901,E2 -1295.901} C_VEL
LIN {X 0,Y 587.319,Z 39.325,A -85,B 0,C 180,E1 -1298.481,E2 -1298.481} C_VEL
LIN {X 0,Y 587.329,Z 39.319,A -85,B 0,C 180,E1 -1301.158,E2 -1301.158} C_VEL
LIN {X 0,Y 587.304,Z 39.328,A -85,B 0,C 180,E1 -1304.112,E2 -1304.112} C_VEL
LIN {X 0,Y 587.303,Z 39.324,A -85,B 0,C 180,E1 -1306.993,E2 -1306.993} C_VEL
LIN {X 0,Y 587.303,Z 39.331,A -85,B 0,C 180,E1 -1309.745,E2 -1309.745} C_VEL
LIN {X 0,Y 587.313,Z 39.322,A -85,B 0,C 180,E1 -1312.39,E2 -1312.39} C_VEL
LIN {X 0,Y 587.338,Z 39.325,A -85,B 0,C 180,E1 -1315.655,E2 -1315.655} C_VEL
LIN {X 0,Y 587.36,Z 39.488,A -85,B 0,C 180,E1 -1318.534,E2 -1318.534} C_VEL
LIN {X 0,Y 587.342,Z 53.226,A -85,B 0,C 180,E1 -1321.134,E2 -1321.134} C_VEL
LIN {X 0,Y 587.326,Z 60.861,A -85,B 0,C 180,E1 -1322.565,E2 -1322.565} C_VEL
LIN {X 0,Y 587.877,Z 65.87,A -85,B 0,C 180,E1 -1322.647,E2 -1322.647} C_VEL
LIN {X 0,Y 587.747,Z 167.358,A -85,B 0,C 180,E1 -1323.908,E2 -1323.908} C_VEL
LIN {X 0,Y 587.684,Z 180.537,A -85,B 0,C 180,E1 -1324.215,E2 -1324.215} C_VEL
LIN {X 0,Y 587.587,Z 192.841,A -85,B 0,C 180,E1 -1324.638,E2 -1324.638} C_VEL
LIN {X 0,Y 587.533,Z 204.07,A -85,B 0,C 180,E1 -1325.156,E2 -1325.156} C_VEL
LIN {X 0,Y 587.395,Z 215.422,A -85,B 0,C 180,E1 -1325.828,E2 -1325.828} C_VEL
LIN {X 0,Y 587.379,Z 226.455,A -85,B 0,C 180,E1 -1326.651,E2 -1326.651} C_VEL
LIN {X 0,Y 587.328,Z 235.553,A -85,B 0,C 180,E1 -1327.486,E2 -1327.486} C_VEL
LIN {X 0,Y 587.274,Z 243.767,A -85,B 0,C 180,E1 -1328.409,E2 -1328.409} C_VEL
LIN {X 0,Y 587.219,Z 251.689,A -85,B 0,C 180,E1 -1329.509,E2 -1329.509} C_VEL
LIN {X 0,Y 587.191,Z 256.995,A -85,B 0,C 180,E1 -1330.42,E2 -1330.42} C_VEL
LIN {X 0,Y 587.174,Z 262.061,A -85,B 0,C 180,E1 -1331.508,E2 -1331.508} C_VEL
LIN {X 0,Y 587.163,Z 265.88,A -85,B 0,C 180,E1 -1332.589,E2 -1332.589} C_VEL
LIN {X 0,Y 587.15,Z 267.822,A -85,B 0,C 180,E1 -1333.306,E2 -1333.306} C_VEL
LIN {X 0,Y 587.139,Z 269.254,A -85,B 0,C 180,E1 -1334.02,E2 -1334.02} C_VEL
LIN {X 0,Y 587.125,Z 270.253,A -85,B 0,C 180,E1 -1334.732,E2 -1334.732} C_VEL
LIN {X 0,Y 587.162,Z 270.955,A -85,B 0,C 180,E1 -1335.82,E2 -1335.82} C_VEL
LIN {X 0,Y 587.146,Z 270.701,A -85,B 0,C 180,E1 -1336.855,E2 -1336.855} C_VEL
LIN {X 0,Y 587.161,Z 270.021,A -85,B 0,C 180,E1 -1337.558,E2 -1337.558} C_VEL
LIN {X 0,Y 587.155,Z 268.928,A -85,B 0,C 180,E1 -1338.26,E2 -1338.26} C_VEL
LIN {X 0,Y 587.168,Z 267.373,A -85,B 0,C 180,E1 -1338.959,E2 -1338.959} C_VEL
LIN {X 0,Y 587.179,Z 264.243,A -85,B 0,C 180,E1 -1340.006,E2 -1340.006} C_VEL
LIN {X 0,Y 587.186,Z 260.051,A -85,B 0,C 180,E1 -1341.049,E2 -1341.049} C_VEL
LIN {X 0,Y 587.232,Z 253.668,A -85,B 0,C 180,E1 -1342.262,E2 -1342.262} C_VEL
LIN {X 0,Y 587.24,Z 246.104,A -85,B 0,C 180,E1 -1343.384,E2 -1343.384} C_VEL
LIN {X 0,Y 587.29,Z 238.102,A -85,B 0,C 180,E1 -1344.334,E2 -1344.334} C_VEL
LIN {X 0,Y 587.388,Z 229.275,A -85,B 0,C 180,E1 -1345.196,E2 -1345.196} C_VEL
LIN {X 0,Y 587.459,Z 218.446,A -85,B 0,C 180,E1 -1346.056,E2 -1346.056} C_VEL
LIN {X 0,Y 587.532,Z 207.548,A -85,B 0,C 180,E1 -1346.743,E2 -1346.743} C_VEL
LIN {X 0,Y 587.581,Z 195.422,A -85,B 0,C 180,E1 -1347.344,E2 -1347.344} C_VEL
LIN {X 0,Y 587.61,Z 183.993,A -85,B 0,C 180,E1 -1347.773,E2 -1347.773} C_VEL
LIN {X 0,Y 587.671,Z 171.964,A -85,B 0,C 180,E1 -1348.094,E2 -1348.094} C_VEL
LIN {X 0,Y 587.749,Z 156.772,A -85,B 0,C 180,E1 -1348.33,E2 -1348.33} C_VEL
LIN {X 0,Y 587.72,Z 63.516,A -85,B 0,C 180,E1 -1349.476,E2 -1349.476} C_VEL
LIN {X 0,Y 587.289,Z 60.843,A -85,B 0,C 180,E1 -1349.529,E2 -1349.529} C_VEL
LIN {X 0,Y 587.38,Z 47.378,A -85,B 0,C 180,E1 -1352.057,E2 -1352.057} C_VEL
LIN {X 0,Y 587.376,Z 39.317,A -85,B 0,C 180,E1 -1353.602,E2 -1353.602} C_VEL
LIN {X 0,Y 587.38,Z 39.323,A -85,B 0,C 180,E1 -1356.733,E2 -1356.733} C_VEL
LIN {X 0,Y 587.33,Z 39.324,A -85,B 0,C 180,E1 -1358.949,E2 -1358.949} C_VEL
LIN {X 0,Y 587.335,Z 39.319,A -85,B 0,C 180,E1 -1361.737,E2 -1361.737} C_VEL
LIN {X 0,Y 587.345,Z 39.325,A -85,B 0,C 180,E1 -1364.553,E2 -1364.553} C_VEL
LIN {X 0,Y 587.348,Z 39.317,A -85,B 0,C 180,E1 -1367.406,E2 -1367.406} C_VEL
LIN {X 0,Y 587.33,Z 39.328,A -85,B 0,C 180,E1 -1370.305,E2 -1370.305} C_VEL
LIN {X 0,Y 587.319,Z 39.321,A -85,B 0,C 180,E1 -1373.259,E2 -1373.259} C_VEL
LIN {X 0,Y 587.334,Z 39.321,A -85,B 0,C 180,E1 -1375.517,E2 -1375.517} C_VEL
LIN {X 0,Y 587.351,Z 39.324,A -85,B 0,C 180,E1 -1377.818,E2 -1377.818} C_VEL
LIN {X 0,Y 587.341,Z 39.319,A -85,B 0,C 180,E1 -1380.51,E2 -1380.51} C_VEL
LIN {X 0,Y 587.337,Z 39.322,A -85,B 0,C 180,E1 -1383.397,E2 -1383.397} C_VEL
LIN {X 0,Y 587.298,Z 39.329,A -85,B 0,C 180,E1 -1385.9,E2 -1385.9} C_VEL
LIN {X 0,Y 587.325,Z 39.32,A -85,B 0,C 180,E1 -1388.48,E2 -1388.48} C_VEL
LIN {X 0,Y 587.339,Z 39.322,A -85,B 0,C 180,E1 -1391.157,E2 -1391.157} C_VEL
LIN {X 0,Y 587.316,Z 39.322,A -85,B 0,C 180,E1 -1394.112,E2 -1394.112} C_VEL
LIN {X 0,Y 587.316,Z 39.326,A -85,B 0,C 180,E1 -1396.993,E2 -1396.993} C_VEL
LIN {X 0,Y 587.318,Z 39.323,A -85,B 0,C 180,E1 -1399.745,E2 -1399.745} C_VEL
LIN {X 0,Y 587.347,Z 39.318,A -85,B 0,C 180,E1 -1402.392,E2 -1402.392} C_VEL
LIN {X 0,Y 587.35,Z 39.318,A -85,B 0,C 180,E1 -1405.652,E2 -1405.652} C_VEL
LIN {X 0,Y 587.341,Z 39.319,A -85,B 0,C 180,E1 -1408.231,E2 -1408.231} C_VEL
LIN {X 0,Y 587.351,Z 39.326,A -85,B 0,C 180,E1 -1410.867,E2 -1410.867} C_VEL
LIN {X 0,Y 587.34,Z 39.318,A -85,B 0,C 180,E1 -1413.721,E2 -1413.721} C_VEL
LIN {X 0,Y 587.339,Z 39.319,A -85,B 0,C 180,E1 -1415.993,E2 -1415.993} C_VEL
LIN {X 0,Y 587.327,Z 39.324,A -85,B 0,C 180,E1 -1418.226,E2 -1418.226} C_VEL
LIN {X 0,Y 587.349,Z 39.318,A -85,B 0,C 180,E1 -1421.151,E2 -1421.151} C_VEL
LIN {X 0,Y 587.324,Z 39.325,A -85,B 0,C 180,E1 -1424.025,E2 -1424.025} C_VEL
LIN {X 0,Y 587.359,Z 39.323,A -85,B 0,C 180,E1 -1426.154,E2 -1426.154} C_VEL
LIN {X 0,Y 587.343,Z 39.318,A -85,B 0,C 180,E1 -1428.962,E2 -1428.962} C_VEL
LIN {X 0,Y 587.368,Z 39.319,A -85,B 0,C 180,E1 -1431.745,E2 -1431.745} C_VEL
LIN {X 0,Y 587.352,Z 39.319,A -85,B 0,C 180,E1 -1434.507,E2 -1434.507} C_VEL
LIN {X 0,Y 587.374,Z 39.315,A -85,B 0,C 180,E1 -1437.257,E2 -1437.257} C_VEL
LIN {X 0,Y 587.381,Z 39.319,A -85,B 0,C 180,E1 -1440,E2 -1440} C_VEL
LIN {X 0,Y 587.37,Z 39.314,A -85,B 0,C 180,E1 -1442.743,E2 -1442.743} C_VEL
LIN {X 0,Y 587.355,Z 39.324,A -85,B 0,C 180,E1 -1445.493,E2 -1445.493} C_VEL
LIN {X 0,Y 587.342,Z 39.318,A -85,B 0,C 180,E1 -1448.255,E2 -1448.255} C_VEL
LIN {X 0,Y 587.351,Z 39.322,A -85,B 0,C 180,E1 -1451.134,E2 -1451.134} C_VEL
LIN {X 0,Y 587.359,Z 39.315,A -85,B 0,C 180,E1 -1454.257,E2 -1454.257} C_VEL
LIN {X 0,Y 587.349,Z 39.323,A -85,B 0,C 180,E1 -1457.406,E2 -1457.406} C_VEL
LIN {X 0,Y 587.329,Z 39.32,A -85,B 0,C 180,E1 -1460.305,E2 -1460.305} C_VEL
LIN {X 0,Y 587.314,Z 39.326,A -85,B 0,C 180,E1 -1463.259,E2 -1463.259} C_VEL
LIN {X 0,Y 587.325,Z 39.321,A -85,B 0,C 180,E1 -1465.517,E2 -1465.517} C_VEL
LIN {X 0,Y 587.309,Z 39.322,A -85,B 0,C 180,E1 -1467.82,E2 -1467.82} C_VEL
LIN {X 0,Y 587.337,Z 39.325,A -85,B 0,C 180,E1 -1470.51,E2 -1470.51} C_VEL
LIN {X 0,Y 587.329,Z 39.32,A -85,B 0,C 180,E1 -1473.397,E2 -1473.397} C_VEL
LIN {X 0,Y 587.298,Z 39.324,A -85,B 0,C 180,E1 -1475.9,E2 -1475.9} C_VEL
LIN {X 0,Y 587.328,Z 39.329,A -85,B 0,C 180,E1 -1478.48,E2 -1478.48} C_VEL
LIN {X 0,Y 587.335,Z 39.319,A -85,B 0,C 180,E1 -1481.157,E2 -1481.157} C_VEL
LIN {X 0,Y 587.314,Z 39.329,A -85,B 0,C 180,E1 -1484.112,E2 -1484.112} C_VEL
LIN {X 0,Y 587.313,Z 39.321,A -85,B 0,C 180,E1 -1486.993,E2 -1486.993} C_VEL
LIN {X 0,Y 587.313,Z 39.326,A -85,B 0,C 180,E1 -1489.745,E2 -1489.745} C_VEL
LIN {X 0,Y 587.344,Z 39.321,A -85,B 0,C 180,E1 -1492.392,E2 -1492.392} C_VEL
LIN {X 0,Y 587.347,Z 39.324,A -85,B 0,C 180,E1 -1495.653,E2 -1495.653} C_VEL
LIN {X 0,Y 587.342,Z 39.32,A -85,B 0,C 180,E1 -1498.231,E2 -1498.231} C_VEL
LIN {X 0,Y 587.351,Z 39.318,A -85,B 0,C 180,E1 -1500.867,E2 -1500.867} C_VEL
LIN {X 0,Y 587.339,Z 39.325,A -85,B 0,C 180,E1 -1503.824,E2 -1503.824} C_VEL
LIN {X 0,Y 587.363,Z 39.487,A -85,B 0,C 180,E1 -1506.112,E2 -1506.112} C_VEL
LIN {X 0,Y 587.878,Z 44.216,A -85,B 0,C 180,E1 -1506.764,E2 -1506.764} C_VEL
LIN {X 0,Y 587.749,Z 66.573,A -85,B 0,C 180,E1 -1509.71,E2 -1509.71} C_VEL
LIN {X 0,Y 587.634,Z 89.624,A -85,B 0,C 180,E1 -1512.762,E2 -1512.762} C_VEL
LIN {X 0,Y 587.457,Z 111.762,A -85,B 0,C 180,E1 -1515.645,E2 -1515.645} C_VEL
LIN {X 0,Y 587.4,Z 118.353,A -85,B 0,C 180,E1 -1516.497,E2 -1516.497} C_VEL
LIN {X 0,Y 587.847,Z 122.701,A -85,B 0,C 180,E1 -1516.562,E2 -1516.562} C_VEL
LIN {X 0,Y 587.725,Z 226.935,A -85,B 0,C 180,E1 -1517.855,E2 -1517.855} C_VEL
LIN {X 0,Y 587.671,Z 240.211,A -85,B 0,C 180,E1 -1518.16,E2 -1518.16} C_VEL
LIN {X 0,Y 587.615,Z 252.636,A -85,B 0,C 180,E1 -1518.585,E2 -1518.585} C_VEL
LIN {X 0,Y 587.558,Z 264.624,A -85,B 0,C 180,E1 -1519.141,E2 -1519.141} C_VEL
LIN {X 0,Y 587.458,Z 276.199,A -85,B 0,C 180,E1 -1519.836,E2 -1519.836} C_VEL
LIN {X 0,Y 587.366,Z 286.597,A -85,B 0,C 180,E1 -1520.617,E2 -1520.617} C_VEL
LIN {X 0,Y 587.322,Z 295.11,A -85,B 0,C 180,E1 -1521.397,E2 -1521.397} C_VEL
LIN {X 0,Y 587.274,Z 302.959,A -85,B 0,C 180,E1 -1522.263,E2 -1522.263} C_VEL
LIN {X 0,Y 587.23,Z 309.467,A -85,B 0,C 180,E1 -1523.126,E2 -1523.126} C_VEL
LIN {X 0,Y 587.237,Z 315.865,A -85,B 0,C 180,E1 -1524.161,E2 -1524.161} C_VEL
LIN {X 0,Y 587.147,Z 320.949,A -85,B 0,C 180,E1 -1525.193,E2 -1525.193} C_VEL
LIN {X 0,Y 587.213,Z 324.895,A -85,B 0,C 180,E1 -1526.225,E2 -1526.225} C_VEL
LIN {X 0,Y 587.132,Z 327.808,A -85,B 0,C 180,E1 -1527.255,E2 -1527.255} C_VEL
LIN {X 0,Y 587.141,Z 329.199,A -85,B 0,C 180,E1 -1527.942,E2 -1527.942} C_VEL
LIN {X 0,Y 587.14,Z 330.785,A -85,B 0,C 180,E1 -1529.314,E2 -1529.314} C_VEL
LIN {X 0,Y 587.137,Z 331,A -85,B 0,C 180,E1 -1530,E2 -1530} C_VEL
LIN {X 0,Y 587.147,Z 330.186,A -85,B 0,C 180,E1 -1531.372,E2 -1531.372} C_VEL
LIN {X 0,Y 587.141,Z 329.201,A -85,B 0,C 180,E1 -1532.058,E2 -1532.058} C_VEL
LIN {X 0,Y 587.132,Z 327.81,A -85,B 0,C 180,E1 -1532.744,E2 -1532.744} C_VEL
LIN {X 0,Y 587.213,Z 324.897,A -85,B 0,C 180,E1 -1533.774,E2 -1533.774} C_VEL
LIN {X 0,Y 587.147,Z 320.95,A -85,B 0,C 180,E1 -1534.806,E2 -1534.806} C_VEL
LIN {X 0,Y 587.218,Z 314.879,A -85,B 0,C 180,E1 -1536.011,E2 -1536.011} C_VEL
LIN {X 0,Y 587.244,Z 308.239,A -85,B 0,C 180,E1 -1537.046,E2 -1537.046} C_VEL
LIN {X 0,Y 587.299,Z 299.993,A -85,B 0,C 180,E1 -1538.083,E2 -1538.083} C_VEL
LIN {X 0,Y 587.343,Z 291.541,A -85,B 0,C 180,E1 -1538.949,E2 -1538.949} C_VEL
LIN {X 0,Y 587.413,Z 281.101,A -85,B 0,C 180,E1 -1539.816,E2 -1539.816} C_VEL
LIN {X 0,Y 587.48,Z 270.76,A -85,B 0,C 180,E1 -1540.511,E2 -1540.511} C_VEL
LIN {X 0,Y 587.582,Z 258.819,A -85,B 0,C 180,E1 -1541.148,E2 -1541.148} C_VEL
LIN {X 0,Y 587.63,Z 246.605,A -85,B 0,C 180,E1 -1541.639,E2 -1541.639} C_VEL
LIN {X 0,Y 587.701,Z 233.446,A -85,B 0,C 180,E1 -1542.014,E2 -1542.014} C_VEL
LIN {X 0,Y 587.773,Z 221.105,A -85,B 0,C 180,E1 -1542.231,E2 -1542.231} C_VEL
LIN {X 0,Y 587.726,Z 120.507,A -85,B 0,C 180,E1 -1543.468,E2 -1543.468} C_VEL
LIN {X 0,Y 587.408,Z 118.272,A -85,B 0,C 180,E1 -1543.514,E2 -1543.514} C_VEL
LIN {X 0,Y 587.546,Z 96.606,A -85,B 0,C 180,E1 -1546.325,E2 -1546.325} C_VEL
LIN {X 0,Y 587.667,Z 77.5,A -85,B 0,C 180,E1 -1548.838,E2 -1548.838} C_VEL
LIN {X 0,Y 587.795,Z 58.13,A -85,B 0,C 180,E1 -1551.395,E2 -1551.395} C_VEL
LIN {X 0,Y 587.865,Z 42.786,A -85,B 0,C 180,E1 -1553.422,E2 -1553.422} C_VEL
LIN {X 0,Y 587.347,Z 39.324,A -85,B 0,C 180,E1 -1553.912,E2 -1553.912} C_VEL
LIN {X 0,Y 587.338,Z 39.327,A -85,B 0,C 180,E1 -1556.278,E2 -1556.278} C_VEL
LIN {X 0,Y 587.35,Z 39.318,A -85,B 0,C 180,E1 -1559.133,E2 -1559.133} C_VEL
LIN {X 0,Y 587.344,Z 39.323,A -85,B 0,C 180,E1 -1561.835,E2 -1561.835} C_VEL
LIN {X 0,Y 587.35,Z 39.322,A -85,B 0,C 180,E1 -1564.348,E2 -1564.348} C_VEL
LIN {X 0,Y 587.353,Z 39.317,A -85,B 0,C 180,E1 -1566.746,E2 -1566.746} C_VEL
LIN {X 0,Y 587.332,Z 39.322,A -85,B 0,C 180,E1 -1569.36,E2 -1569.36} C_VEL
LIN {X 0,Y 587.334,Z 39.323,A -85,B 0,C 180,E1 -1572.107,E2 -1572.107} C_VEL
LIN {X 0,Y 587.304,Z 39.324,A -85,B 0,C 180,E1 -1575.087,E2 -1575.087} C_VEL
LIN {X 0,Y 587.352,Z 39.32,A -85,B 0,C 180,E1 -1577.927,E2 -1577.927} C_VEL
LIN {X 0,Y 587.331,Z 39.324,A -85,B 0,C 180,E1 -1581.058,E2 -1581.058} C_VEL
LIN {X 0,Y 587.352,Z 39.326,A -85,B 0,C 180,E1 -1583.291,E2 -1583.291} C_VEL
LIN {X 0,Y 587.367,Z 39.316,A -85,B 0,C 180,E1 -1585.78,E2 -1585.78} C_VEL
LIN {X 0,Y 587.344,Z 39.318,A -85,B 0,C 180,E1 -1588.231,E2 -1588.231} C_VEL
LIN {X 0,Y 587.347,Z 39.325,A -85,B 0,C 180,E1 -1590.866,E2 -1590.866} C_VEL
LIN {X 0,Y 587.357,Z 39.316,A -85,B 0,C 180,E1 -1593.819,E2 -1593.819} C_VEL
LIN {X 0,Y 587.336,Z 39.319,A -85,B 0,C 180,E1 -1595.993,E2 -1595.993} C_VEL
LIN {X 0,Y 587.323,Z 39.323,A -85,B 0,C 180,E1 -1598.226,E2 -1598.226} C_VEL
LIN {X 0,Y 587.347,Z 39.318,A -85,B 0,C 180,E1 -1601.151,E2 -1601.151} C_VEL
LIN {X 0,Y 587.323,Z 39.324,A -85,B 0,C 180,E1 -1604.025,E2 -1604.025} C_VEL
LIN {X 0,Y 587.356,Z 39.323,A -85,B 0,C 180,E1 -1606.154,E2 -1606.154} C_VEL
LIN {X 0,Y 587.34,Z 39.319,A -85,B 0,C 180,E1 -1608.963,E2 -1608.963} C_VEL
LIN {X 0,Y 587.369,Z 39.319,A -85,B 0,C 180,E1 -1611.745,E2 -1611.745} C_VEL
LIN {X 0,Y 587.35,Z 39.319,A -85,B 0,C 180,E1 -1614.507,E2 -1614.507} C_VEL
LIN {X 0,Y 587.373,Z 39.315,A -85,B 0,C 180,E1 -1617.257,E2 -1617.257} C_VEL
LIN {X 0,Y 587.377,Z 39.319,A -85,B 0,C 180,E1 -1620,E2 -1620} C_VEL
LIN {X 0,Y 587.367,Z 39.314,A -85,B 0,C 180,E1 -1622.743,E2 -1622.743} C_VEL
LIN {X 0,Y 587.354,Z 39.326,A -85,B 0,C 180,E1 -1625.493,E2 -1625.493} C_VEL
LIN {X 0,Y 587.326,Z 39.319,A -85,B 0,C 180,E1 -1628.256,E2 -1628.256} C_VEL
LIN {X 0,Y 587.346,Z 39.325,A -85,B 0,C 180,E1 -1631.134,E2 -1631.134} C_VEL
LIN {X 0,Y 587.354,Z 39.316,A -85,B 0,C 180,E1 -1634.257,E2 -1634.257} C_VEL
LIN {X 0,Y 587.343,Z 39.321,A -85,B 0,C 180,E1 -1637.406,E2 -1637.406} C_VEL
LIN {X 0,Y 587.3,Z 39.324,A -85,B 0,C 180,E1 -1638.306,E2 -1638.306} C_VEL
LIN {X 0,Y 586.663,Z 39.411,A -85,B 0,C 180,E1 -1638.878,E2 -1638.878} C_VEL
LIN {X 0,Y 583.843,Z 39.763,A -85,B 0,C 180,E1 -1639.807,E2 -1639.807} C_VEL
LIN {X 0,Y 581.432,Z 40.062,A -85,B 0,C 180,E1 -1640.554,E2 -1640.554} C_VEL
LIN {X 0,Y 580.377,Z 40.19,A -85,B 0,C 180,E1 -1641.13,E2 -1641.13} C_VEL
LIN {X 0,Y 580.281,Z 40.199,A -85,B 0,C 180,E1 -1641.325,E2 -1641.325} C_VEL
LIN {X 0,Y 580.295,Z 40.2,A -85,B 0,C 180,E1 -1644.317,E2 -1644.317} C_VEL
LIN {X 0,Y 580.262,Z 40.209,A -85,B 0,C 180,E1 -1646.624,E2 -1646.624} C_VEL
LIN {X 0,Y 580.295,Z 40.196,A -85,B 0,C 180,E1 -1649.309,E2 -1649.309} C_VEL
LIN {X 0,Y 580.296,Z 40.202,A -85,B 0,C 180,E1 -1652.201,E2 -1652.201} C_VEL
LIN {X 0,Y 580.276,Z 40.201,A -85,B 0,C 180,E1 -1654.698,E2 -1654.698} C_VEL
LIN {X 0,Y 580.286,Z 40.197,A -85,B 0,C 180,E1 -1657.27,E2 -1657.27} C_VEL
LIN {X 0,Y 580.285,Z 40.202,A -85,B 0,C 180,E1 -1660.27,E2 -1660.27} C_VEL
LIN {X 0,Y 580.252,Z 40.203,A -85,B 0,C 180,E1 -1662.709,E2 -1662.709} C_VEL
LIN {X 0,Y 580.25,Z 40.208,A -85,B 0,C 180,E1 -1665.612,E2 -1665.612} C_VEL
LIN {X 0,Y 580.253,Z 40.204,A -85,B 0,C 180,E1 -1668.229,E2 -1668.229} C_VEL
LIN {X 0,Y 580.263,Z 40.202,A -85,B 0,C 180,E1 -1670.964,E2 -1670.964} C_VEL
LIN {X 0,Y 580.245,Z 40.211,A -85,B 0,C 180,E1 -1673.595,E2 -1673.595} C_VEL
LIN {X 0,Y 580.276,Z 40.201,A -85,B 0,C 180,E1 -1676.143,E2 -1676.143} C_VEL
LIN {X 0,Y 580.306,Z 40.328,A -85,B 0,C 180,E1 -1678.465,E2 -1678.465} C_VEL
LIN {X 0,Y 580.327,Z 51.847,A -85,B 0,C 180,E1 -1680.687,E2 -1680.687} C_VEL
LIN {X 0,Y 580.29,Z 60.841,A -85,B 0,C 180,E1 -1682.395,E2 -1682.395} C_VEL
LIN {X 0,Y 580.978,Z 66.225,A -85,B 0,C 180,E1 -1682.489,E2 -1682.489} C_VEL
LIN {X 0,Y 580.834,Z 167.138,A -85,B 0,C 180,E1 -1683.757,E2 -1683.757} C_VEL
LIN {X 0,Y 580.739,Z 180.413,A -85,B 0,C 180,E1 -1684.068,E2 -1684.068} C_VEL
LIN {X 0,Y 580.636,Z 192.971,A -85,B 0,C 180,E1 -1684.504,E2 -1684.504} C_VEL
LIN {X 0,Y 580.546,Z 204.201,A -85,B 0,C 180,E1 -1685.03,E2 -1685.03} C_VEL
LIN {X 0,Y 580.39,Z 215.201,A -85,B 0,C 180,E1 -1685.688,E2 -1685.688} C_VEL
LIN {X 0,Y 580.378,Z 225.371,A -85,B 0,C 180,E1 -1686.447,E2 -1686.447} C_VEL
LIN {X 0,Y 580.295,Z 235.597,A -85,B 0,C 180,E1 -1687.386,E2 -1687.386} C_VEL
LIN {X 0,Y 580.221,Z 243.802,A -85,B 0,C 180,E1 -1688.32,E2 -1688.32} C_VEL
LIN {X 0,Y 580.137,Z 251.714,A -85,B 0,C 180,E1 -1689.432,E2 -1689.432} C_VEL
LIN {X 0,Y 580.1,Z 257.97,A -85,B 0,C 180,E1 -1690.539,E2 -1690.539} C_VEL
LIN {X 0,Y 580.075,Z 262.82,A -85,B 0,C 180,E1 -1691.639,E2 -1691.639} C_VEL
LIN {X 0,Y 580.055,Z 266.44,A -85,B 0,C 180,E1 -1692.732,E2 -1692.732} C_VEL
LIN {X 0,Y 580.034,Z 268.96,A -85,B 0,C 180,E1 -1693.819,E2 -1693.819} C_VEL
LIN {X 0,Y 580.021,Z 270.052,A -85,B 0,C 180,E1 -1694.54,E2 -1694.54} C_VEL
LIN {X 0,Y 580.053,Z 270.944,A -85,B 0,C 180,E1 -1695.766,E2 -1695.766} C_VEL
LIN {X 0,Y 580.061,Z 270.817,A -85,B 0,C 180,E1 -1696.691,E2 -1696.691} C_VEL
LIN {X 0,Y 580.051,Z 270.22,A -85,B 0,C 180,E1 -1697.403,E2 -1697.403} C_VEL
LIN {X 0,Y 580.055,Z 269.22,A -85,B 0,C 180,E1 -1698.114,E2 -1698.114} C_VEL
LIN {X 0,Y 580.076,Z 267.552,A -85,B 0,C 180,E1 -1698.925,E2 -1698.925} C_VEL
LIN {X 0,Y 580.083,Z 263.602,A -85,B 0,C 180,E1 -1700.235,E2 -1700.235} C_VEL
LIN {X 0,Y 580.112,Z 259.217,A -85,B 0,C 180,E1 -1701.29,E2 -1701.29} C_VEL
LIN {X 0,Y 580.145,Z 253.647,A -85,B 0,C 180,E1 -1702.342,E2 -1702.342} C_VEL
LIN {X 0,Y 580.185,Z 246.897,A -85,B 0,C 180,E1 -1703.367,E2 -1703.367} C_VEL
LIN {X 0,Y 580.212,Z 239.67,A -85,B 0,C 180,E1 -1704.265,E2 -1704.265} C_VEL
LIN {X 0,Y 580.311,Z 231.169,A -85,B 0,C 180,E1 -1705.137,E2 -1705.137} C_VEL
LIN {X 0,Y 580.397,Z 220.743,A -85,B 0,C 180,E1 -1706.008,E2 -1706.008} C_VEL
LIN {X 0,Y 580.507,Z 210.44,A -85,B 0,C 180,E1 -1706.704,E2 -1706.704} C_VEL
LIN {X 0,Y 580.607,Z 199.182,A -85,B 0,C 180,E1 -1707.312,E2 -1707.312} C_VEL
LIN {X 0,Y 580.617,Z 187.71,A -85,B 0,C 180,E1 -1707.789,E2 -1707.789} C_VEL
LIN {X 0,Y 580.746,Z 174.481,A -85,B 0,C 180,E1 -1708.18,E2 -1708.18} C_VEL
LIN {X 0,Y 580.813,Z 161.567,A -85,B 0,C 180,E1 -1708.418,E2 -1708.418} C_VEL
LIN {X 0,Y 580.768,Z 64.125,A -85,B 0,C 180,E1 -1709.632,E2 -1709.632} C_VEL
LIN {X 0,Y 580.25,Z 60.838,A -85,B 0,C 180,E1 -1709.697,E2 -1709.697} C_VEL
LIN {X 0,Y 580.435,Z 44.662,A -85,B 0,C 180,E1 -1712.776,E2 -1712.776} C_VEL
LIN {X 0,Y 580.305,Z 40.199,A -85,B 0,C 180,E1 -1713.689,E2 -1713.689} C_VEL
LIN {X 0,Y 580.287,Z 40.2,A -85,B 0,C 180,E1 -1716.258,E2 -1716.258} C_VEL
LIN {X 0,Y 580.333,Z 40.197,A -85,B 0,C 180,E1 -1718.356,E2 -1718.356} C_VEL
LIN {X 0,Y 580.307,Z 40.195,A -85,B 0,C 180,E1 -1721.191,E2 -1721.191} C_VEL
LIN {X 0,Y 580.329,Z 40.194,A -85,B 0,C 180,E1 -1724.017,E2 -1724.017} C_VEL
LIN {X 0,Y 580.32,Z 40.194,A -85,B 0,C 180,E1 -1726.914,E2 -1726.914} C_VEL
LIN {X 0,Y 580.291,Z 40.199,A -85,B 0,C 180,E1 -1729.823,E2 -1729.823} C_VEL
LIN {X 0,Y 580.277,Z 40.206,A -85,B 0,C 180,E1 -1732.053,E2 -1732.053} C_VEL
LIN {X 0,Y 580.31,Z 40.194,A -85,B 0,C 180,E1 -1735.08,E2 -1735.08} C_VEL
LIN {X 0,Y 580.301,Z 40.201,A -85,B 0,C 180,E1 -1738.186,E2 -1738.186} C_VEL
LIN {X 0,Y 580.289,Z 40.196,A -85,B 0,C 180,E1 -1740.694,E2 -1740.694} C_VEL
LIN {X 0,Y 580.307,Z 40.197,A -85,B 0,C 180,E1 -1743.316,E2 -1743.316} C_VEL
LIN {X 0,Y 580.265,Z 40.208,A -85,B 0,C 180,E1 -1745.758,E2 -1745.758} C_VEL
LIN {X 0,Y 580.289,Z 40.198,A -85,B 0,C 180,E1 -1748.147,E2 -1748.147} C_VEL
LIN {X 0,Y 580.301,Z 40.196,A -85,B 0,C 180,E1 -1750.843,E2 -1750.843} C_VEL
LIN {X 0,Y 580.277,Z 40.204,A -85,B 0,C 180,E1 -1753.658,E2 -1753.658} C_VEL
LIN {X 0,Y 580.277,Z 40.199,A -85,B 0,C 180,E1 -1756.61,E2 -1756.61} C_VEL
LIN {X 0,Y 580.301,Z 40.204,A -85,B 0,C 180,E1 -1759.156,E2 -1759.156} C_VEL
LIN {X 0,Y 580.291,Z 40.196,A -85,B 0,C 180,E1 -1761.927,E2 -1761.927} C_VEL
LIN {X 0,Y 580.256,Z 40.202,A -85,B 0,C 180,E1 -1764.453,E2 -1764.453} C_VEL
LIN {X 0,Y 580.291,Z 40.206,A -85,B 0,C 180,E1 -1766.975,E2 -1766.975} C_VEL
LIN {X 0,Y 580.299,Z 40.197,A -85,B 0,C 180,E1 -1769.425,E2 -1769.425} C_VEL
LIN {X 0,Y 580.3,Z 40.196,A -85,B 0,C 180,E1 -1772.141,E2 -1772.141} C_VEL
LIN {X 0,Y 580.325,Z 40.193,A -85,B 0,C 180,E1 -1775.27,E2 -1775.27} C_VEL
LIN {X 0,Y 580.277,Z 40.199,A -85,B 0,C 180,E1 -1777.947,E2 -1777.947} C_VEL
LIN {X 0,Y 580.302,Z 40.198,A -85,B 0,C 180,E1 -1780.913,E2 -1780.913} C_VEL
LIN {X 0,Y 580.279,Z 40.2,A -85,B 0,C 180,E1 -1783.825,E2 -1783.825} C_VEL
LIN {X 0,Y 580.327,Z 40.196,A -85,B 0,C 180,E1 -1785.983,E2 -1785.983} C_VEL
LIN {X 0,Y 580.308,Z 40.195,A -85,B 0,C 180,E1 -1788.827,E2 -1788.827} C_VEL
LIN {X 0,Y 580.33,Z 40.194,A -85,B 0,C 180,E1 -1791.644,E2 -1791.644} C_VEL
LIN {X 0,Y 580.319,Z 40.195,A -85,B 0,C 180,E1 -1794.44,E2 -1794.44} C_VEL
LIN {X 0,Y 580.34,Z 40.191,A -85,B 0,C 180,E1 -1797.223,E2 -1797.223} C_VEL
LIN {X 0,Y 580.351,Z 40.195,A -85,B 0,C 180,E1 -1800,E2 -1800} C_VEL
LIN {X 0,Y 580.336,Z 40.19,A -85,B 0,C 180,E1 -1802.776,E2 -1802.776} C_VEL
LIN {X 0,Y 580.32,Z 40.202,A -85,B 0,C 180,E1 -1805.56,E2 -1805.56} C_VEL
LIN {X 0,Y 580.325,Z 40.199,A -85,B 0,C 180,E1 -1807.655,E2 -1807.655} C_VEL
LIN {X 0,Y 580.299,Z 40.195,A -85,B 0,C 180,E1 -1810.467,E2 -1810.467} C_VEL
LIN {X 0,Y 580.275,Z 40.208,A -85,B 0,C 180,E1 -1813.304,E2 -1813.304} C_VEL
LIN {X 0,Y 580.295,Z 40.202,A -85,B 0,C 180,E1 -1815.453,E2 -1815.453} C_VEL
LIN {X 0,Y 580.291,Z 40.199,A -85,B 0,C 180,E1 -1817.625,E2 -1817.625} C_VEL
LIN {X 0,Y 580.289,Z 40.197,A -85,B 0,C 180,E1 -1819.823,E2 -1819.823} C_VEL
LIN {X 0,Y 580.271,Z 40.198,A -85,B 0,C 180,E1 -1822.053,E2 -1822.053} C_VEL
LIN {X 0,Y 580.303,Z 40.201,A -85,B 0,C 180,E1 -1825.08,E2 -1825.08} C_VEL
LIN {X 0,Y 580.285,Z 40.198,A -85,B 0,C 180,E1 -1828.186,E2 -1828.186} C_VEL
LIN {X 0,Y 580.285,Z 40.207,A -85,B 0,C 180,E1 -1830.694,E2 -1830.694} C_VEL
LIN {X 0,Y 580.285,Z 40.198,A -85,B 0,C 180,E1 -1833.313,E2 -1833.313} C_VEL
LIN {X 0,Y 580.252,Z 40.201,A -85,B 0,C 180,E1 -1835.757,E2 -1835.757} C_VEL
LIN {X 0,Y 580.289,Z 40.201,A -85,B 0,C 180,E1 -1838.146,E2 -1838.146} C_VEL
LIN {X 0,Y 580.297,Z 40.198,A -85,B 0,C 180,E1 -1840.844,E2 -1840.844} C_VEL
LIN {X 0,Y 580.275,Z 40.2,A -85,B 0,C 180,E1 -1843.658,E2 -1843.658} C_VEL
LIN {X 0,Y 580.275,Z 40.201,A -85,B 0,C 180,E1 -1846.61,E2 -1846.61} C_VEL
LIN {X 0,Y 580.298,Z 40.195,A -85,B 0,C 180,E1 -1849.156,E2 -1849.156} C_VEL
LIN {X 0,Y 580.29,Z 40.206,A -85,B 0,C 180,E1 -1851.927,E2 -1851.927} C_VEL
LIN {X 0,Y 580.254,Z 40.202,A -85,B 0,C 180,E1 -1854.453,E2 -1854.453} C_VEL
LIN {X 0,Y 580.291,Z 40.196,A -85,B 0,C 180,E1 -1856.975,E2 -1856.975} C_VEL
LIN {X 0,Y 580.29,Z 40.201,A -85,B 0,C 180,E1 -1859.425,E2 -1859.425} C_VEL
LIN {X 0,Y 580.295,Z 40.199,A -85,B 0,C 180,E1 -1862.142,E2 -1862.142} C_VEL
LIN {X 0,Y 580.322,Z 40.2,A -85,B 0,C 180,E1 -1865.27,E2 -1865.27} C_VEL
LIN {X 0,Y 580.332,Z 40.369,A -85,B 0,C 180,E1 -1865.97,E2 -1865.97} C_VEL
LIN {X 0,Y 580.94,Z 45.839,A -85,B 0,C 180,E1 -1866.735,E2 -1866.735} C_VEL
LIN {X 0,Y 580.769,Z 67.616,A -85,B 0,C 180,E1 -1869.64,E2 -1869.64} C_VEL
LIN {X 0,Y 580.657,Z 89.915,A -85,B 0,C 180,E1 -1872.587,E2 -1872.587} C_VEL
LIN {X 0,Y 580.435,Z 110.25,A -85,B 0,C 180,E1 -1875.269,E2 -1875.269} C_VEL
LIN {X 0,Y 580.422,Z 118.353,A -85,B 0,C 180,E1 -1876.331,E2 -1876.331} C_VEL
LIN {X 0,Y 580.95,Z 124.49,A -85,B 0,C 180,E1 -1876.422,E2 -1876.422} C_VEL
LIN {X 0,Y 580.785,Z 226.934,A -85,B 0,C 180,E1 -1877.707,E2 -1877.707} C_VEL
LIN {X 0,Y 580.741,Z 240.21,A -85,B 0,C 180,E1 -1878.017,E2 -1878.017} C_VEL
LIN {X 0,Y 580.656,Z 252.37,A -85,B 0,C 180,E1 -1878.436,E2 -1878.436} C_VEL
LIN {X 0,Y 580.58,Z 264.622,A -85,B 0,C 180,E1 -1879.009,E2 -1879.009} C_VEL
LIN {X 0,Y 580.436,Z 276.196,A -85,B 0,C 180,E1 -1879.712,E2 -1879.712} C_VEL
LIN {X 0,Y 580.346,Z 286.599,A -85,B 0,C 180,E1 -1880.503,E2 -1880.503} C_VEL
LIN {X 0,Y 580.271,Z 295.11,A -85,B 0,C 180,E1 -1881.292,E2 -1881.292} C_VEL
LIN {X 0,Y 580.222,Z 302.959,A -85,B 0,C 180,E1 -1882.168,E2 -1882.168} C_VEL
LIN {X 0,Y 580.154,Z 310.65,A -85,B 0,C 180,E1 -1883.221,E2 -1883.221} C_VEL
LIN {X 0,Y 580.139,Z 317.679,A -85,B 0,C 180,E1 -1884.438,E2 -1884.438} C_VEL
LIN {X 0,Y 580.108,Z 322.371,A -85,B 0,C 180,E1 -1885.483,E2 -1885.483} C_VEL
LIN {X 0,Y 580.123,Z 325.957,A -85,B 0,C 180,E1 -1886.527,E2 -1886.527} C_VEL
LIN {X 0,Y 580.043,Z 327.807,A -85,B 0,C 180,E1 -1887.222,E2 -1887.222} C_VEL
LIN {X 0,Y 580.04,Z 329.197,A -85,B 0,C 180,E1 -1887.917,E2 -1887.917} C_VEL
LIN {X 0,Y 580.04,Z 330.785,A -85,B 0,C 180,E1 -1889.306,E2 -1889.306} C_VEL
LIN {X 0,Y 580.037,Z 331,A -85,B 0,C 180,E1 -1890,E2 -1890} C_VEL
LIN {X 0,Y 580.046,Z 330.186,A -85,B 0,C 180,E1 -1891.388,E2 -1891.388} C_VEL
LIN {X 0,Y 580.04,Z 329.199,A -85,B 0,C 180,E1 -1892.083,E2 -1892.083} C_VEL
LIN {X 0,Y 580.043,Z 327.811,A -85,B 0,C 180,E1 -1892.778,E2 -1892.778} C_VEL
LIN {X 0,Y 580.11,Z 324.897,A -85,B 0,C 180,E1 -1893.82,E2 -1893.82} C_VEL
LIN {X 0,Y 580.053,Z 320.95,A -85,B 0,C 180,E1 -1894.865,E2 -1894.865} C_VEL
LIN {X 0,Y 580.139,Z 314.878,A -85,B 0,C 180,E1 -1896.085,E2 -1896.085} C_VEL
LIN {X 0,Y 580.184,Z 308.239,A -85,B 0,C 180,E1 -1897.132,E2 -1897.132} C_VEL
LIN {X 0,Y 580.25,Z 299.993,A -85,B 0,C 180,E1 -1898.182,E2 -1898.182} C_VEL
LIN {X 0,Y 580.308,Z 291.542,A -85,B 0,C 180,E1 -1899.058,E2 -1899.058} C_VEL
LIN {X 0,Y 580.416,Z 281.101,A -85,B 0,C 180,E1 -1899.936,E2 -1899.936} C_VEL
LIN {X 0,Y 580.501,Z 270.758,A -85,B 0,C 180,E1 -1900.639,E2 -1900.639} C_VEL
LIN {X 0,Y 580.596,Z 259.248,A -85,B 0,C 180,E1 -1901.264,E2 -1901.264} C_VEL
LIN {X 0,Y 580.669,Z 246.48,A -85,B 0,C 180,E1 -1901.785,E2 -1901.785} C_VEL
LIN {X 0,Y 580.775,Z 233.444,A -85,B 0,C 180,E1 -1902.159,E2 -1902.159} C_VEL
LIN {X 0,Y 580.857,Z 221.105,A -85,B 0,C 180,E1 -1902.379,E2 -1902.379} C_VEL
LIN {X 0,Y 580.818,Z 121.179,A -85,B 0,C 180,E1 -1903.622,E2 -1903.622} C_VEL
LIN {X 0,Y 580.429,Z 118.272,A -85,B 0,C 180,E1 -1903.679,E2 -1903.679} C_VEL
LIN {X 0,Y 580.599,Z 95.242,A -85,B 0,C 180,E1 -1906.707,E2 -1906.707} C_VEL
LIN {X 0,Y 580.701,Z 77.374,A -85,B 0,C 180,E1 -1909.073,E2 -1909.073} C_VEL
LIN {X 0,Y 580.819,Z 57.8,A -85,B 0,C 180,E1 -1911.657,E2 -1911.657} C_VEL
LIN {X 0,Y 580.895,Z 43.821,A -85,B 0,C 180,E1 -1913.531,E2 -1913.531} C_VEL
LIN {X 0,Y 580.312,Z 40.202,A -85,B 0,C 180,E1 -1914.078,E2 -1914.078} C_VEL
LIN {X 0,Y 580.278,Z 40.205,A -85,B 0,C 180,E1 -1916.623,E2 -1916.623} C_VEL
LIN {X 0,Y 580.301,Z 40.196,A -85,B 0,C 180,E1 -1919.309,E2 -1919.309} C_VEL
LIN {X 0,Y 580.298,Z 40.205,A -85,B 0,C 180,E1 -1922.2,E2 -1922.2} C_VEL
LIN {X 0,Y 580.299,Z 40.196,A -85,B 0,C 180,E1 -1924.695,E2 -1924.695} C_VEL
LIN {X 0,Y 580.299,Z 40.196,A -85,B 0,C 180,E1 -1927.268,E2 -1927.268} C_VEL
LIN {X 0,Y 580.292,Z 40.2,A -85,B 0,C 180,E1 -1930.27,E2 -1930.27} C_VEL
LIN {X 0,Y 580.276,Z 40.198,A -85,B 0,C 180,E1 -1932.706,E2 -1932.706} C_VEL
LIN {X 0,Y 580.266,Z 40.207,A -85,B 0,C 180,E1 -1935.609,E2 -1935.609} C_VEL
LIN {X 0,Y 580.297,Z 40.196,A -85,B 0,C 180,E1 -1938.233,E2 -1938.233} C_VEL
LIN {X 0,Y 580.287,Z 40.2,A -85,B 0,C 180,E1 -1940.966,E2 -1940.966} C_VEL
LIN {X 0,Y 580.295,Z 40.2,A -85,B 0,C 180,E1 -1943.598,E2 -1943.598} C_VEL
LIN {X 0,Y 580.318,Z 40.192,A -85,B 0,C 180,E1 -1946.145,E2 -1946.145} C_VEL
LIN {X 0,Y 580.28,Z 40.201,A -85,B 0,C 180,E1 -1948.615,E2 -1948.615} C_VEL
LIN {X 0,Y 580.291,Z 40.205,A -85,B 0,C 180,E1 -1951.024,E2 -1951.024} C_VEL
LIN {X 0,Y 580.29,Z 40.196,A -85,B 0,C 180,E1 -1953.666,E2 -1953.666} C_VEL
LIN {X 0,Y 580.299,Z 40.195,A -85,B 0,C 180,E1 -1955.684,E2 -1955.684} C_VEL
LIN {X 0,Y 580.273,Z 40.198,A -85,B 0,C 180,E1 -1957.947,E2 -1957.947} C_VEL
LIN {X 0,Y 580.317,Z 40.196,A -85,B 0,C 180,E1 -1960.914,E2 -1960.914} C_VEL
LIN {X 0,Y 580.278,Z 40.199,A -85,B 0,C 180,E1 -1963.826,E2 -1963.826} C_VEL
LIN {X 0,Y 580.323,Z 40.197,A -85,B 0,C 180,E1 -1965.983,E2 -1965.983} C_VEL
LIN {X 0,Y 580.302,Z 40.196,A -85,B 0,C 180,E1 -1968.827,E2 -1968.827} C_VEL
LIN {X 0,Y 580.333,Z 40.194,A -85,B 0,C 180,E1 -1971.644,E2 -1971.644} C_VEL
LIN {X 0,Y 580.317,Z 40.196,A -85,B 0,C 180,E1 -1974.44,E2 -1974.44} C_VEL
LIN {X 0,Y 580.338,Z 40.191,A -85,B 0,C 180,E1 -1977.224,E2 -1977.224} C_VEL
LIN {X 0,Y 580.346,Z 40.195,A -85,B 0,C 180,E1 -1980,E2 -1980} C_VEL
LIN {X 0,Y 580.334,Z 40.19,A -85,B 0,C 180,E1 -1982.777,E2 -1982.777} C_VEL
LIN {X 0,Y 580.319,Z 40.202,A -85,B 0,C 180,E1 -1985.56,E2 -1985.56} C_VEL
LIN {X 0,Y 580.316,Z 40.198,A -85,B 0,C 180,E1 -1987.656,E2 -1987.656} C_VEL
LIN {X 0,Y 580.295,Z 40.196,A -85,B 0,C 180,E1 -1990.467,E2 -1990.467} C_VEL
LIN {X 0,Y 580.271,Z 40.206,A -85,B 0,C 180,E1 -1993.304,E2 -1993.304} C_VEL
LIN {X 0,Y 580.291,Z 40.2,A -85,B 0,C 180,E1 -1995.453,E2 -1995.453} C_VEL
LIN {X 0,Y 580.286,Z 40.197,A -85,B 0,C 180,E1 -1997.625,E2 -1997.625} C_VEL
LIN {X 0,Y 580.285,Z 40.197,A -85,B 0,C 180,E1 -1999.823,E2 -1999.823} C_VEL
LIN {X 0,Y 580.281,Z 40.199,A -85,B 0,C 180,E1 -2001.325,E2 -2001.325} C_VEL
LIN {X 0,Y 579.581,Z 40.286,A -85,B 0,C 180,E1 -2001.905,E2 -2001.905} C_VEL
LIN {X 0,Y 576.702,Z 40.652,A -85,B 0,C 180,E1 -2002.844,E2 -2002.844} C_VEL
LIN {X 0,Y 574.308,Z 40.946,A -85,B 0,C 180,E1 -2003.601,E2 -2003.601} C_VEL
LIN {X 0,Y 573.31,Z 41.069,A -85,B 0,C 180,E1 -2004.184,E2 -2004.184} C_VEL
LIN {X 0,Y 573.244,Z 41.079,A -85,B 0,C 180,E1 -2004.382,E2 -2004.382} C_VEL
LIN {X 0,Y 573.199,Z 41.084,A -85,B 0,C 180,E1 -2006.979,E2 -2006.979} C_VEL
LIN {X 0,Y 573.241,Z 41.074,A -85,B 0,C 180,E1 -2009.488,E2 -2009.488} C_VEL
LIN {X 0,Y 573.251,Z 41.078,A -85,B 0,C 180,E1 -2012.646,E2 -2012.646} C_VEL
LIN {X 0,Y 573.192,Z 41.08,A -85,B 0,C 180,E1 -2015.189,E2 -2015.189} C_VEL
LIN {X 0,Y 573.229,Z 41.081,A -85,B 0,C 180,E1 -2017.809,E2 -2017.809} C_VEL
LIN {X 0,Y 573.245,Z 41.075,A -85,B 0,C 180,E1 -2020.526,E2 -2020.526} C_VEL
LIN {X 0,Y 573.199,Z 41.083,A -85,B 0,C 180,E1 -2023.363,E2 -2023.363} C_VEL
LIN {X 0,Y 573.21,Z 41.082,A -85,B 0,C 180,E1 -2026.335,E2 -2026.335} C_VEL
LIN {X 0,Y 573.205,Z 41.079,A -85,B 0,C 180,E1 -2028.541,E2 -2028.541} C_VEL
LIN {X 0,Y 573.23,Z 41.082,A -85,B 0,C 180,E1 -2031.298,E2 -2031.298} C_VEL
LIN {X 0,Y 573.189,Z 41.084,A -85,B 0,C 180,E1 -2034.023,E2 -2034.023} C_VEL
LIN {X 0,Y 573.225,Z 41.079,A -85,B 0,C 180,E1 -2036.515,E2 -2036.515} C_VEL
LIN {X 0,Y 573.265,Z 41.243,A -85,B 0,C 180,E1 -2038.393,E2 -2038.393} C_VEL
LIN {X 0,Y 573.327,Z 52.022,A -85,B 0,C 180,E1 -2040.499,E2 -2040.499} C_VEL
LIN {X 0,Y 573.245,Z 60.889,A -85,B 0,C 180,E1 -2042.233,E2 -2042.233} C_VEL
LIN {X 0,Y 574.098,Z 66.519,A -85,B 0,C 180,E1 -2042.327,E2 -2042.327} C_VEL
LIN {X 0,Y 573.899,Z 167.424,A -85,B 0,C 180,E1 -2043.612,E2 -2043.612} C_VEL
LIN {X 0,Y 573.801,Z 180.877,A -85,B 0,C 180,E1 -2043.935,E2 -2043.935} C_VEL
LIN {X 0,Y 573.694,Z 193.105,A -85,B 0,C 180,E1 -2044.368,E2 -2044.368} C_VEL
LIN {X 0,Y 573.552,Z 205.221,A -85,B 0,C 180,E1 -2044.951,E2 -2044.951} C_VEL
LIN {X 0,Y 573.359,Z 216.644,A -85,B 0,C 180,E1 -2045.66,E2 -2045.66} C_VEL
LIN {X 0,Y 573.328,Z 227.684,A -85,B 0,C 180,E1 -2046.523,E2 -2046.523} C_VEL
LIN {X 0,Y 573.199,Z 237.376,A -85,B 0,C 180,E1 -2047.471,E2 -2047.471} C_VEL
LIN {X 0,Y 573.129,Z 245.273,A -85,B 0,C 180,E1 -2048.416,E2 -2048.416} C_VEL
LIN {X 0,Y 573.075,Z 252.917,A -85,B 0,C 180,E1 -2049.543,E2 -2049.543} C_VEL
LIN {X 0,Y 573.005,Z 259.555,A -85,B 0,C 180,E1 -2050.809,E2 -2050.809} C_VEL
LIN {X 0,Y 572.988,Z 264.79,A -85,B 0,C 180,E1 -2052.144,E2 -2052.144} C_VEL
LIN {X 0,Y 572.947,Z 267.468,A -85,B 0,C 180,E1 -2053.095,E2 -2053.095} C_VEL
LIN {X 0,Y 572.917,Z 269.84,A -85,B 0,C 180,E1 -2054.343,E2 -2054.343} C_VEL
LIN {X 0,Y 572.946,Z 270.931,A -85,B 0,C 180,E1 -2055.709,E2 -2055.709} C_VEL
LIN {X 0,Y 572.971,Z 270.898,A -85,B 0,C 180,E1 -2056.523,E2 -2056.523} C_VEL
LIN {X 0,Y 572.947,Z 270.415,A -85,B 0,C 180,E1 -2057.245,E2 -2057.245} C_VEL
LIN {X 0,Y 572.948,Z 269.499,A -85,B 0,C 180,E1 -2057.964,E2 -2057.964} C_VEL
LIN {X 0,Y 572.99,Z 267.738,A -85,B 0,C 180,E1 -2058.886,E2 -2058.886} C_VEL
LIN {X 0,Y 573.005,Z 264.213,A -85,B 0,C 180,E1 -2060.113,E2 -2060.113} C_VEL
LIN {X 0,Y 573.025,Z 260.011,A -85,B 0,C 180,E1 -2061.182,E2 -2061.182} C_VEL
LIN {X 0,Y 573.073,Z 253.624,A -85,B 0,C 180,E1 -2062.425,E2 -2062.425} C_VEL
LIN {X 0,Y 573.134,Z 246.021,A -85,B 0,C 180,E1 -2063.576,E2 -2063.576} C_VEL
LIN {X 0,Y 573.186,Z 238.032,A -85,B 0,C 180,E1 -2064.548,E2 -2064.548} C_VEL
LIN {X 0,Y 573.28,Z 229.199,A -85,B 0,C 180,E1 -2065.43,E2 -2065.43} C_VEL
LIN {X 0,Y 573.408,Z 218.347,A -85,B 0,C 180,E1 -2066.311,E2 -2066.311} C_VEL
LIN {X 0,Y 573.55,Z 207.406,A -85,B 0,C 180,E1 -2067.015,E2 -2067.015} C_VEL
LIN {X 0,Y 573.637,Z 195.234,A -85,B 0,C 180,E1 -2067.63,E2 -2067.63} C_VEL
LIN {X 0,Y 573.716,Z 183.729,A -85,B 0,C 180,E1 -2068.07,E2 -2068.07} C_VEL
LIN {X 0,Y 573.832,Z 171.487,A -85,B 0,C 180,E1 -2068.399,E2 -2068.399} C_VEL
LIN {X 0,Y 573.915,Z 155.995,A -85,B 0,C 180,E1 -2068.641,E2 -2068.641} C_VEL
LIN {X 0,Y 573.961,Z 65.329,A -85,B 0,C 180,E1 -2069.781,E2 -2069.781} C_VEL
LIN {X 0,Y 573.207,Z 60.833,A -85,B 0,C 180,E1 -2069.869,E2 -2069.869} C_VEL
LIN {X 0,Y 573.421,Z 45.744,A -85,B 0,C 180,E1 -2072.81,E2 -2072.81} C_VEL
LIN {X 0,Y 573.251,Z 41.078,A -85,B 0,C 180,E1 -2073.779,E2 -2073.779} C_VEL
LIN {X 0,Y 573.25,Z 41.078,A -85,B 0,C 180,E1 -2076.335,E2 -2076.335} C_VEL
LIN {X 0,Y 573.288,Z 41.076,A -85,B 0,C 180,E1 -2078.46,E2 -2078.46} C_VEL
LIN {X 0,Y 573.279,Z 41.07,A -85,B 0,C 180,E1 -2081.312,E2 -2081.312} C_VEL
LIN {X 0,Y 573.288,Z 41.078,A -85,B 0,C 180,E1 -2084.424,E2 -2084.424} C_VEL
LIN {X 0,Y 573.265,Z 41.072,A -85,B 0,C 180,E1 -2087.112,E2 -2087.112} C_VEL
LIN {X 0,Y 573.246,Z 41.081,A -85,B 0,C 180,E1 -2090.077,E2 -2090.077} C_VEL
LIN {X 0,Y 573.24,Z 41.081,A -85,B 0,C 180,E1 -2092.338,E2 -2092.338} C_VEL
LIN {X 0,Y 573.254,Z 41.074,A -85,B 0,C 180,E1 -2095.41,E2 -2095.41} C_VEL
LIN {X 0,Y 573.255,Z 41.081,A -85,B 0,C 180,E1 -2098.028,E2 -2098.028} C_VEL
LIN {X 0,Y 573.233,Z 41.075,A -85,B 0,C 180,E1 -2100.882,E2 -2100.882} C_VEL
LIN {X 0,Y 573.268,Z 41.076,A -85,B 0,C 180,E1 -2103.524,E2 -2103.524} C_VEL
LIN {X 0,Y 573.243,Z 41.078,A -85,B 0,C 180,E1 -2106.05,E2 -2106.05} C_VEL
LIN {X 0,Y 573.243,Z 41.074,A -85,B 0,C 180,E1 -2108.702,E2 -2108.702} C_VEL
LIN {X 0,Y 573.234,Z 41.083,A -85,B 0,C 180,E1 -2111.593,E2 -2111.593} C_VEL
LIN {X 0,Y 573.226,Z 41.076,A -85,B 0,C 180,E1 -2114.335,E2 -2114.335} C_VEL
LIN {X 0,Y 573.244,Z 41.083,A -85,B 0,C 180,E1 -2117.358,E2 -2117.358} C_VEL
LIN {X 0,Y 573.25,Z 41.073,A -85,B 0,C 180,E1 -2120.393,E2 -2120.393} C_VEL
LIN {X 0,Y 573.256,Z 41.082,A -85,B 0,C 180,E1 -2123.077,E2 -2123.077} C_VEL
LIN {X 0,Y 573.27,Z 41.072,A -85,B 0,C 180,E1 -2125.671,E2 -2125.671} C_VEL
LIN {X 0,Y 573.242,Z 41.075,A -85,B 0,C 180,E1 -2128.184,E2 -2128.184} C_VEL
LIN {X 0,Y 573.267,Z 41.078,A -85,B 0,C 180,E1 -2130.634,E2 -2130.634} C_VEL
LIN {X 0,Y 573.253,Z 41.078,A -85,B 0,C 180,E1 -2133.024,E2 -2133.024} C_VEL
LIN {X 0,Y 573.278,Z 41.07,A -85,B 0,C 180,E1 -2135.366,E2 -2135.366} C_VEL
LIN {X 0,Y 573.233,Z 41.083,A -85,B 0,C 180,E1 -2138.419,E2 -2138.419} C_VEL
LIN {X 0,Y 573.272,Z 41.076,A -85,B 0,C 180,E1 -2140.731,E2 -2140.731} C_VEL
LIN {X 0,Y 573.251,Z 41.074,A -85,B 0,C 180,E1 -2143.621,E2 -2143.621} C_VEL
LIN {X 0,Y 573.275,Z 41.073,A -85,B 0,C 180,E1 -2145.807,E2 -2145.807} C_VEL
LIN {X 0,Y 573.266,Z 41.073,A -85,B 0,C 180,E1 -2148.745,E2 -2148.745} C_VEL
LIN {X 0,Y 573.286,Z 41.071,A -85,B 0,C 180,E1 -2151.54,E2 -2151.54} C_VEL
LIN {X 0,Y 573.287,Z 41.072,A -85,B 0,C 180,E1 -2154.372,E2 -2154.372} C_VEL
LIN {X 0,Y 573.308,Z 41.075,A -85,B 0,C 180,E1 -2157.892,E2 -2157.892} C_VEL
LIN {X 0,Y 573.33,Z 41.063,A -85,B 0,C 180,E1 -2160.702,E2 -2160.702} C_VEL
LIN {X 0,Y 573.234,Z 41.082,A -85,B 0,C 180,E1 -2163.514,E2 -2163.514} C_VEL
LIN {X 0,Y 573.287,Z 41.078,A -85,B 0,C 180,E1 -2165.628,E2 -2165.628} C_VEL
LIN {X 0,Y 573.273,Z 41.076,A -85,B 0,C 180,E1 -2167.75,E2 -2167.75} C_VEL
LIN {X 0,Y 573.266,Z 41.071,A -85,B 0,C 180,E1 -2170.597,E2 -2170.597} C_VEL
LIN {X 0,Y 573.265,Z 41.073,A -85,B 0,C 180,E1 -2172.748,E2 -2172.748} C_VEL
LIN {X 0,Y 573.236,Z 41.079,A -85,B 0,C 180,E1 -2174.92,E2 -2174.92} C_VEL
LIN {X 0,Y 573.242,Z 41.075,A -85,B 0,C 180,E1 -2177.849,E2 -2177.849} C_VEL
LIN {X 0,Y 573.244,Z 41.074,A -85,B 0,C 180,E1 -2180.077,E2 -2180.077} C_VEL
LIN {X 0,Y 573.235,Z 41.076,A -85,B 0,C 180,E1 -2182.338,E2 -2182.338} C_VEL
LIN {X 0,Y 573.247,Z 41.076,A -85,B 0,C 180,E1 -2185.41,E2 -2185.41} C_VEL
LIN {X 0,Y 573.232,Z 41.081,A -85,B 0,C 180,E1 -2188.565,E2 -2188.565} C_VEL
LIN {X 0,Y 573.226,Z 41.081,A -85,B 0,C 180,E1 -2190.993,E2 -2190.993} C_VEL
LIN {X 0,Y 573.265,Z 41.071,A -85,B 0,C 180,E1 -2193.524,E2 -2193.524} C_VEL
LIN {X 0,Y 573.218,Z 41.08,A -85,B 0,C 180,E1 -2196.051,E2 -2196.051} C_VEL
LIN {X 0,Y 573.242,Z 41.079,A -85,B 0,C 180,E1 -2198.702,E2 -2198.702} C_VEL
LIN {X 0,Y 573.231,Z 41.076,A -85,B 0,C 180,E1 -2201.593,E2 -2201.593} C_VEL
LIN {X 0,Y 573.224,Z 41.084,A -85,B 0,C 180,E1 -2204.335,E2 -2204.335} C_VEL
LIN {X 0,Y 573.241,Z 41.075,A -85,B 0,C 180,E1 -2207.359,E2 -2207.359} C_VEL
LIN {X 0,Y 573.239,Z 41.078,A -85,B 0,C 180,E1 -2210.392,E2 -2210.392} C_VEL
LIN {X 0,Y 573.254,Z 41.073,A -85,B 0,C 180,E1 -2213.077,E2 -2213.077} C_VEL
LIN {X 0,Y 573.268,Z 41.078,A -85,B 0,C 180,E1 -2215.671,E2 -2215.671} C_VEL
LIN {X 0,Y 573.241,Z 41.077,A -85,B 0,C 180,E1 -2218.184,E2 -2218.184} C_VEL
LIN {X 0,Y 573.262,Z 41.073,A -85,B 0,C 180,E1 -2220.634,E2 -2220.634} C_VEL
LIN {X 0,Y 573.238,Z 41.085,A -85,B 0,C 180,E1 -2223.508,E2 -2223.508} C_VEL
LIN {X 0,Y 573.297,Z 41.251,A -85,B 0,C 180,E1 -2225.825,E2 -2225.825} C_VEL
LIN {X 0,Y 573.987,Z 45.801,A -85,B 0,C 180,E1 -2226.477,E2 -2226.477} C_VEL
LIN {X 0,Y 573.825,Z 64.637,A -85,B 0,C 180,E1 -2229.031,E2 -2229.031} C_VEL
LIN {X 0,Y 573.697,Z 85.382,A -85,B 0,C 180,E1 -2231.797,E2 -2231.797} C_VEL
LIN {X 0,Y 573.52,Z 106.156,A -85,B 0,C 180,E1 -2234.542,E2 -2234.542} C_VEL
LIN {X 0,Y 573.439,Z 118.353,A -85,B 0,C 180,E1 -2236.162,E2 -2236.162} C_VEL
LIN {X 0,Y 574.047,Z 124.49,A -85,B 0,C 180,E1 -2236.256,E2 -2236.256} C_VEL
LIN {X 0,Y 573.85,Z 226.934,A -85,B 0,C 180,E1 -2237.557,E2 -2237.557} C_VEL
LIN {X 0,Y 573.802,Z 240.21,A -85,B 0,C 180,E1 -2237.87,E2 -2237.87} C_VEL
LIN {X 0,Y 573.71,Z 252.372,A -85,B 0,C 180,E1 -2238.294,E2 -2238.294} C_VEL
LIN {X 0,Y 573.586,Z 264.658,A -85,B 0,C 180,E1 -2238.875,E2 -2238.875} C_VEL
LIN {X 0,Y 573.425,Z 276.193,A -85,B 0,C 180,E1 -2239.585,E2 -2239.585} C_VEL
LIN {X 0,Y 573.333,Z 286.601,A -85,B 0,C 180,E1 -2240.385,E2 -2240.385} C_VEL
LIN {X 0,Y 573.241,Z 295.111,A -85,B 0,C 180,E1 -2241.184,E2 -2241.184} C_VEL
LIN {X 0,Y 573.161,Z 302.959,A -85,B 0,C 180,E1 -2242.071,E2 -2242.071} C_VEL
LIN {X 0,Y 573.073,Z 310.954,A -85,B 0,C 180,E1 -2243.185,E2 -2243.185} C_VEL
LIN {X 0,Y 573.07,Z 317.678,A -85,B 0,C 180,E1 -2244.369,E2 -2244.369} C_VEL
LIN {X 0,Y 573.028,Z 322.371,A -85,B 0,C 180,E1 -2245.427,E2 -2245.427} C_VEL
LIN {X 0,Y 573.022,Z 325.957,A -85,B 0,C 180,E1 -2246.484,E2 -2246.484} C_VEL
LIN {X 0,Y 572.959,Z 327.807,A -85,B 0,C 180,E1 -2247.187,E2 -2247.187} C_VEL
LIN {X 0,Y 572.946,Z 330.184,A -85,B 0,C 180,E1 -2248.594,E2 -2248.594} C_VEL
LIN {X 0,Y 572.938,Z 331,A -85,B 0,C 180,E1 -2250,E2 -2250} C_VEL
LIN {X 0,Y 572.946,Z 330.186,A -85,B 0,C 180,E1 -2251.406,E2 -2251.406} C_VEL
LIN {X 0,Y 572.959,Z 327.811,A -85,B 0,C 180,E1 -2252.812,E2 -2252.812} C_VEL
LIN {X 0,Y 573.014,Z 324.896,A -85,B 0,C 180,E1 -2253.868,E2 -2253.868} C_VEL
LIN {X 0,Y 572.963,Z 320.95,A -85,B 0,C 180,E1 -2254.925,E2 -2254.925} C_VEL
LIN {X 0,Y 573.093,Z 315.868,A -85,B 0,C 180,E1 -2255.983,E2 -2255.983} C_VEL
LIN {X 0,Y 573.103,Z 309.469,A -85,B 0,C 180,E1 -2257.044,E2 -2257.044} C_VEL
LIN {X 0,Y 573.177,Z 301.48,A -85,B 0,C 180,E1 -2258.106,E2 -2258.106} C_VEL
LIN {X 0,Y 573.254,Z 293.337,A -85,B 0,C 180,E1 -2258.993,E2 -2258.993} C_VEL
LIN {X 0,Y 573.344,Z 283.402,A -85,B 0,C 180,E1 -2259.881,E2 -2259.881} C_VEL
LIN {X 0,Y 573.501,Z 272.19,A -85,B 0,C 180,E1 -2260.681,E2 -2260.681} C_VEL
LIN {X 0,Y 573.586,Z 261.179,A -85,B 0,C 180,E1 -2261.305,E2 -2261.305} C_VEL
LIN {X 0,Y 573.698,Z 248.987,A -85,B 0,C 180,E1 -2261.84,E2 -2261.84} C_VEL
LIN {X 0,Y 573.811,Z 236.186,A -85,B 0,C 180,E1 -2262.242,E2 -2262.242} C_VEL
LIN {X 0,Y 573.909,Z 222.62,A -85,B 0,C 180,E1 -2262.509,E2 -2262.509} C_VEL
LIN {X 0,Y 573.94,Z 121.973,A -85,B 0,C 180,E1 -2263.779,E2 -2263.779} C_VEL
LIN {X 0,Y 573.441,Z 118.272,A -85,B 0,C 180,E1 -2263.849,E2 -2263.849} C_VEL
LIN {X 0,Y 573.6,Z 96.529,A -85,B 0,C 180,E1 -2266.731,E2 -2266.731} C_VEL
LIN {X 0,Y 573.723,Z 76.359,A -85,B 0,C 180,E1 -2269.397,E2 -2269.397} C_VEL
LIN {X 0,Y 573.892,Z 54.63,A -85,B 0,C 180,E1 -2272.311,E2 -2272.311} C_VEL
LIN {X 0,Y 573.903,Z 44.579,A -85,B 0,C 180,E1 -2273.682,E2 -2273.682} C_VEL
LIN {X 0,Y 573.272,Z 41.08,A -85,B 0,C 180,E1 -2274.2,E2 -2274.2} C_VEL
LIN {X 0,Y 573.252,Z 41.076,A -85,B 0,C 180,E1 -2276.976,E2 -2276.976} C_VEL
LIN {X 0,Y 573.247,Z 41.076,A -85,B 0,C 180,E1 -2279.488,E2 -2279.488} C_VEL
LIN {X 0,Y 573.253,Z 41.076,A -85,B 0,C 180,E1 -2282.645,E2 -2282.645} C_VEL
LIN {X 0,Y 573.267,Z 41.071,A -85,B 0,C 180,E1 -2285.183,E2 -2285.183} C_VEL
LIN {X 0,Y 573.236,Z 41.083,A -85,B 0,C 180,E1 -2287.807,E2 -2287.807} C_VEL
